C09134=1237.357,-18.440,-39.557,-179.564,5.238,148.773
C09135=1237.362,-18.689,-39.544,-179.566,5.238,148.774
C09136=1237.367,-18.939,-39.530,-179.568,5.238,148.775
C09137=1237.372,-19.189,-39.516,-179.571,5.237,148.776
C09138=1237.378,-19.438,-39.502,-179.573,5.237,148.776
C09139=1237.382,-19.687,-39.488,-179.576,5.237,148.777
C09140=1237.387,-19.938,-39.475,-179.578,5.236,148.778
C09141=1237.393,-20.187,-39.461,-179.581,5.237,148.778
C09142=1237.398,-20.436,-39.447,-179.583,5.236,148.779
C09143=1237.402,-20.686,-39.434,-179.585,5.236,148.780
C09144=1237.408,-20.935,-39.420,-179.588,5.236,148.780
C09145=1237.413,-21.185,-39.406,-179.591,5.235,148.781
C09146=1237.418,-21.435,-39.392,-179.593,5.236,148.782
C09147=1237.423,-21.684,-39.379,-179.596,5.236,148.783
C09148=1237.428,-21.954,-39.364,-179.598,5.235,148.783
C09149=1237.434,-22.223,-39.349,-179.601,5.235,148.784
C09150=1237.439,-22.492,-39.334,-179.604,5.235,148.785
C09151=1237.445,-22.761,-39.319,-179.606,5.235,148.786
C09152=1237.449,-23.010,-39.305,-179.609,5.234,148.786
C09153=1237.455,-23.261,-39.292,-179.611,5.234,148.787
C09154=1237.460,-23.510,-39.278,-179.614,5.234,148.788
C09155=1237.464,-23.759,-39.264,-179.616,5.234,148.789
C09156=1237.470,-24.009,-39.251,-179.619,5.234,148.789
C09157=1237.475,-24.259,-39.237,-179.621,5.233,148.790
C09158=1237.480,-24.509,-39.224,-179.623,5.234,148.791
C09159=1237.485,-24.758,-39.210,-179.626,5.233,148.791
C09160=1237.490,-25.007,-39.196,-179.628,5.234,148.792
C09161=1237.495,-25.257,-39.183,-179.631,5.233,148.793
C09162=1237.500,-25.506,-39.169,-179.634,5.233,148.794
C09163=1237.506,-25.757,-39.155,-179.636,5.233,148.794
C09164=1237.510,-26.005,-39.142,-179.639,5.232,148.795
C09165=1237.516,-26.256,-39.128,-179.641,5.233,148.796
C09166=1237.521,-26.504,-39.115,-179.643,5.232,148.796
C09167=1237.526,-26.755,-39.101,-179.646,5.232,148.797
C09168=1237.531,-27.004,-39.087,-179.648,5.232,148.798
C09169=1237.536,-27.253,-39.074,-179.651,5.232,148.799
C09170=1237.541,-27.503,-39.060,-179.653,5.232,148.799
C09171=1237.546,-27.752,-39.047,-179.655,5.231,148.800
C09172=1237.551,-28.002,-39.033,-179.658,5.231,148.801
C09173=1237.557,-28.252,-39.020,-179.661,5.231,148.802
C09174=1237.561,-28.502,-39.006,-179.663,5.231,148.802
C09175=1237.567,-28.751,-38.993,-179.665,5.231,148.803
C09176=1237.571,-29.001,-38.980,-179.668,5.231,148.804
C09177=1237.576,-29.251,-38.966,-179.671,5.230,148.804
C09178=1237.581,-29.500,-38.953,-179.673,5.231,148.805
C09179=1237.586,-29.750,-38.939,-179.675,5.230,148.806
C09180=1237.591,-29.999,-38.926,-179.678,5.230,148.806
C09181=1237.597,-30.249,-38.912,-179.680,5.230,148.807
C09182=1237.601,-30.498,-38.899,-179.683,5.229,148.808
C09183=1237.607,-30.748,-38.885,-179.685,5.230,148.809
C09184=1237.612,-30.998,-38.872,-179.688,5.229,148.809
C09185=1237.617,-31.247,-38.859,-179.690,5.230,148.810
C09186=1237.623,-31.497,-38.845,-179.693,5.229,148.811
C09187=1237.627,-31.746,-38.832,-179.696,5.229,148.812
C09188=1237.633,-31.996,-38.818,-179.698,5.229,148.812
C09189=1237.637,-32.246,-38.805,-179.700,5.229,148.813
C09190=1237.643,-32.495,-38.792,-179.702,5.229,148.814
C09191=1237.647,-32.745,-38.779,-179.705,5.228,148.814
C09192=1237.652,-32.994,-38.766,-179.708,5.228,148.815
C09193=1237.657,-33.244,-38.752,-179.710,5.228,148.816
C09194=1237.662,-33.493,-38.739,-179.712,5.228,148.816
C09195=1237.668,-33.743,-38.726,-179.715,5.228,148.817
C09196=1237.672,-33.992,-38.712,-179.717,5.227,148.818
C09197=1237.678,-34.242,-38.699,-179.720,5.227,148.819
C09198=1237.683,-34.492,-38.686,-179.722,5.228,148.819
C09199=1237.688,-34.741,-38.672,-179.725,5.227,148.820
C09200=1237.693,-34.991,-38.659,-179.727,5.227,148.821
C09201=1237.699,-35.240,-38.646,-179.730,5.227,148.822
C09202=1237.703,-35.490,-38.633,-179.732,5.227,148.822
C09203=1237.708,-35.739,-38.620,-179.735,5.227,148.823
C09204=1237.713,-35.989,-38.606,-179.737,5.226,148.824
C09205=1237.719,-36.239,-38.594,-179.739,5.227,148.824
C09206=1237.724,-36.489,-38.580,-179.742,5.226,148.825
C09207=1237.729,-36.738,-38.567,-179.744,5.226,148.826
C09208=1237.734,-36.987,-38.554,-179.747,5.226,148.826
C09209=1237.739,-37.237,-38.541,-179.749,5.226,148.827
C09210=1237.744,-37.487,-38.528,-179.752,5.226,148.828
C09211=1237.749,-37.737,-38.514,-179.755,5.225,148.829
C09212=1237.754,-37.986,-38.501,-179.757,5.226,148.829
C09213=1237.759,-38.236,-38.488,-179.759,5.225,148.830
C09214=1237.765,-38.485,-38.475,-179.761,5.226,148.831
C09215=1237.770,-38.735,-38.462,-179.764,5.225,148.832
C09216=1237.774,-38.985,-38.449,-179.766,5.225,148.832
C09217=1237.780,-39.234,-38.435,-179.769,5.225,148.833
C09218=1237.784,-39.484,-38.422,-179.772,5.224,148.834
C09219=1237.790,-39.733,-38.409,-179.774,5.225,148.834
C09220=1237.795,-39.983,-38.397,-179.776,5.224,148.835
C09221=1237.800,-40.233,-38.384,-179.778,5.225,148.836
C09222=1237.805,-40.482,-38.371,-179.782,5.224,148.837
C09223=1237.811,-40.732,-38.358,-179.784,5.225,148.837
C09224=1237.815,-40.982,-38.345,-179.786,5.224,148.838
C09225=1237.820,-41.230,-38.332,-179.789,5.224,148.839
C09226=1237.825,-41.481,-38.318,-179.791,5.224,148.840
C09227=1237.831,-41.730,-38.305,-179.794,5.224,148.840
C09228=1237.836,-41.979,-38.293,-179.796,5.224,148.841
C09229=1237.841,-42.230,-38.279,-179.798,5.223,148.842
C09230=1237.846,-42.479,-38.267,-179.801,5.224,148.842
C09231=1237.851,-42.728,-38.254,-179.803,5.223,148.843
C09232=1237.856,-42.978,-38.241,-179.806,5.223,148.844
C09233=1237.862,-43.228,-38.228,-179.808,5.223,148.844
C09234=1237.867,-43.477,-38.215,-179.811,5.223,148.845
C09235=1237.871,-43.727,-38.202,-179.813,5.223,148.846
C09236=1237.876,-43.977,-38.190,-179.816,5.223,148.847
C09237=1237.882,-44.226,-38.177,-179.818,5.223,148.847
C09238=1237.887,-44.476,-38.164,-179.821,5.222,148.848
C09239=1237.892,-44.726,-38.151,-179.823,5.222,148.849
C09240=1237.897,-44.975,-38.138,-179.825,5.222,148.850
C09241=1237.902,-45.225,-38.125,-179.828,5.222,148.850
C09242=1237.907,-45.475,-38.112,-179.830,5.222,148.851
C09243=1237.912,-45.724,-38.100,-179.833,5.222,148.852
C09244=1237.917,-45.974,-38.087,-179.835,5.222,148.852
C09245=1237.922,-46.223,-38.074,-179.838,5.221,148.853
C09246=1237.928,-46.473,-38.061,-179.840,5.222,148.854
C09247=1237.932,-46.723,-38.048,-179.843,5.222,148.855
C09248=1237.938,-46.972,-38.035,-179.845,5.221,148.855
C09249=1237.943,-47.221,-38.023,-179.848,5.221,148.856
C09250=1237.948,-47.471,-38.010,-179.850,5.221,148.857
C09251=1237.953,-47.721,-37.997,-179.852,5.221,148.858
C09252=1237.959,-47.990,-37.983,-179.855,5.221,148.858
C09253=1237.964,-48.260,-37.970,-179.858,5.221,148.859
C09254=1237.970,-48.531,-37.956,-179.860,5.221,148.860
C09255=1237.975,-48.800,-37.943,-179.863,5.220,148.861
C09256=1237.980,-49.050,-37.930,-179.865,5.221,148.861
C09257=1237.985,-49.299,-37.917,-179.868,5.220,148.862
C09258=1237.991,-49.549,-37.904,-179.870,5.220,148.863
C09259=1237.996,-49.798,-37.891,-179.873,5.220,148.864
C09260=1238.001,-50.048,-37.878,-179.876,5.220,148.864
C09261=1238.006,-50.297,-37.866,-179.878,5.220,148.865
C09262=1238.011,-50.547,-37.854,-179.880,5.220,148.866
C09263=1238.016,-50.796,-37.841,-179.882,5.220,148.866
C09264=1238.021,-51.046,-37.828,-179.885,5.220,148.867
C09265=1238.026,-51.296,-37.816,-179.887,5.220,148.868
C09266=1238.031,-51.545,-37.803,-179.890,5.219,148.869
C09267=1238.037,-51.795,-37.791,-179.892,5.220,148.869
C09268=1238.042,-52.045,-37.778,-179.895,5.219,148.870
C09269=1238.047,-52.295,-37.765,-179.897,5.219,148.871
C09270=1238.052,-52.544,-37.752,-179.899,5.219,148.871
C09271=1238.057,-52.793,-37.740,-179.902,5.219,148.872
C09272=1238.062,-53.044,-37.728,-179.905,5.219,148.873
C09273=1238.067,-53.293,-37.715,-179.907,5.219,148.874
C09274=1238.072,-53.543,-37.702,-179.909,5.219,148.874
C09275=1238.077,-53.792,-37.690,-179.912,5.219,148.875
C09276=1238.083,-54.042,-37.678,-179.914,5.219,148.876
C09277=1238.087,-54.292,-37.665,-179.917,5.218,148.877
C09278=1238.092,-54.541,-37.652,-179.919,5.219,148.877
C09279=1238.097,-54.790,-37.640,-179.922,5.218,148.878
C09280=1238.103,-55.040,-37.628,-179.924,5.219,148.879
C09281=1238.108,-55.290,-37.615,-179.926,5.218,148.879
C09282=1238.113,-55.540,-37.602,-179.928,5.218,148.880
C09283=1238.118,-55.790,-37.590,-179.931,5.218,148.881
C09284=1238.123,-56.039,-37.578,-179.934,5.217,148.881
C09285=1238.128,-56.288,-37.565,-179.936,5.218,148.882
C09286=1238.134,-56.538,-37.553,-179.939,5.218,148.883
C09287=1238.139,-56.788,-37.541,-179.941,5.218,148.884
C09288=1238.143,-57.038,-37.528,-179.944,5.218,148.885
C09289=1238.149,-57.288,-37.516,-179.946,5.218,148.885
C09290=1238.154,-57.537,-37.503,-179.948,5.217,148.886
C09291=1238.159,-57.786,-37.491,-179.951,5.218,148.887
C09292=1238.164,-58.036,-37.479,-179.953,5.217,148.887
C09293=1238.169,-58.285,-37.466,-179.955,5.218,148.888
C09294=1238.175,-58.535,-37.454,-179.958,5.217,148.889
C09295=1238.179,-58.785,-37.441,-179.960,5.217,148.889
C09296=1238.185,-59.035,-37.429,-179.963,5.217,148.890
C09297=1238.190,-59.285,-37.417,-179.965,5.217,148.891
C09298=1238.194,-59.534,-37.405,-179.968,5.217,148.892
C09299=1238.200,-59.784,-37.393,-179.971,5.217,148.892
C09300=1238.205,-60.033,-37.380,-179.973,5.217,148.893
C09301=1238.210,-60.283,-37.368,-179.975,5.216,148.894
C09302=1238.215,-60.532,-37.356,-179.977,5.217,148.895
C09303=1238.220,-60.782,-37.343,-179.980,5.216,148.895
C09304=1238.225,-61.032,-37.331,-179.982,5.217,148.896
C09305=1238.231,-61.281,-37.318,-179.985,5.216,148.897
C09306=1238.236,-61.531,-37.306,-179.987,5.216,148.897
C09307=1238.241,-61.781,-37.294,-179.990,5.216,148.898
C09308=1238.246,-62.030,-37.283,-179.992,5.216,148.899
C09309=1238.251,-62.280,-37.270,-179.994,5.216,148.900
C09310=1238.256,-62.530,-37.258,-179.997,5.216,148.900
C09311=1238.261,-62.779,-37.246,-179.999,5.216,148.901
C09312=1238.267,-63.029,-37.234,179.998,5.216,148.902
C09313=1238.272,-63.278,-37.221,179.996,5.216,148.903
C09314=1238.277,-63.529,-37.209,179.993,5.216,148.903
C09315=1238.282,-63.778,-37.197,179.991,5.216,148.904
C09316=1238.287,-64.028,-37.185,179.989,5.216,148.905
C09317=1238.292,-64.278,-37.173,179.986,5.216,148.905
C09318=1238.297,-64.527,-37.160,179.984,5.216,148.906
C09319=1238.303,-64.777,-37.149,179.981,5.215,148.907
C09320=1238.308,-65.026,-37.136,179.979,5.216,148.908
C09321=1238.312,-65.276,-37.125,179.977,5.215,148.908
C09322=1238.318,-65.526,-37.113,179.974,5.216,148.909
C09323=1238.323,-65.775,-37.100,179.972,5.215,148.910
C09324=1238.328,-66.025,-37.088,179.970,5.215,148.910
C09325=1238.334,-66.274,-37.076,179.967,5.215,148.911
C09326=1238.338,-66.524,-37.064,179.964,5.215,148.912
C09327=1238.344,-66.774,-37.052,179.962,5.215,148.913
C09328=1238.349,-67.023,-37.040,179.959,5.215,148.913
C09329=1238.354,-67.273,-37.028,179.957,5.215,148.914
C09330=1238.360,-67.523,-37.016,179.954,5.215,148.915
C09331=1238.364,-67.772,-37.004,179.952,5.215,148.916
C09332=1238.370,-68.022,-36.992,179.950,5.214,148.916
C09333=1238.375,-68.272,-36.980,179.947,5.215,148.917
C09334=1238.380,-68.521,-36.968,179.945,5.214,148.918
C09335=1238.385,-68.771,-36.956,179.943,5.215,148.918
C09336=1238.390,-69.021,-36.945,179.940,5.214,148.919
C09337=1238.395,-69.270,-36.932,179.938,5.214,148.920
C09338=1238.400,-69.520,-36.921,179.935,5.214,148.921
C09339=1238.405,-69.770,-36.909,179.933,5.214,148.921
C09340=1238.411,-70.019,-36.896,179.931,5.214,148.922
C09341=1238.416,-70.269,-36.884,179.928,5.214,148.923
C09342=1238.421,-70.519,-36.873,179.926,5.214,148.923
C09343=1238.426,-70.769,-36.861,179.923,5.214,148.924
C09344=1238.431,-71.018,-36.849,179.921,5.214,148.925
C09345=1238.436,-71.268,-36.837,179.918,5.214,148.926
C09346=1238.441,-71.517,-36.825,179.916,5.214,148.926
C09347=1238.447,-71.767,-36.813,179.914,5.214,148.927
C09348=1238.452,-72.017,-36.801,179.911,5.214,148.928
C09349=1238.457,-72.266,-36.790,179.909,5.214,148.929
C09350=1238.462,-72.516,-36.778,179.906,5.214,148.929
C09351=1238.467,-72.766,-36.766,179.904,5.214,148.930
C09352=1238.472,-73.016,-36.755,179.901,5.213,148.931
C09353=1238.477,-73.265,-36.742,179.899,5.214,148.931
C09354=1238.483,-73.514,-36.730,179.897,5.213,148.932
C09355=1238.488,-73.764,-36.719,179.895,5.214,148.933
C09356=1238.493,-74.034,-36.706,179.891,5.213,148.934
C09357=1238.499,-74.305,-36.693,179.889,5.214,148.934
C09358=1238.505,-74.575,-36.681,179.887,5.213,148.935
C09359=1238.510,-74.845,-36.668,179.884,5.213,148.936
C09360=1238.516,-75.095,-36.656,179.881,5.214,148.937
C09361=1238.520,-75.344,-36.644,179.879,5.213,148.937
C09362=1238.525,-75.594,-36.633,179.877,5.213,148.938
C09363=1238.531,-75.844,-36.621,179.874,5.213,148.939
C09364=1238.536,-76.093,-36.610,179.872,5.213,148.940
C09365=1238.542,-76.343,-36.598,179.869,5.213,148.940
C09366=1238.546,-76.593,-36.587,179.867,5.213,148.941
C09367=1238.552,-76.843,-36.575,179.864,5.213,148.942
C09368=1238.557,-77.093,-36.563,179.862,5.213,148.942
C09369=1238.562,-77.342,-36.551,179.860,5.213,148.943
C09370=1238.567,-77.592,-36.540,179.858,5.213,148.944
C09371=1238.572,-77.842,-36.528,179.855,5.212,148.945
C09372=1238.577,-78.092,-36.516,179.853,5.213,148.945
C09373=1238.582,-78.340,-36.505,179.850,5.212,148.946
C09374=1238.588,-78.590,-36.493,179.848,5.213,148.947
C09375=1238.592,-78.840,-36.482,179.845,5.212,148.947
C09376=1238.598,-79.089,-36.470,179.843,5.213,148.948
C09377=1238.603,-79.339,-36.458,179.841,5.212,148.949
C09378=1238.608,-79.589,-36.447,179.839,5.212,148.950
C09379=1238.613,-79.839,-36.435,179.835,5.212,148.950
C09380=1238.619,-80.088,-36.424,179.833,5.213,148.951
C09381=1238.624,-80.338,-36.412,179.831,5.212,148.952
C09382=1238.629,-80.587,-36.401,179.829,5.213,148.953
C09383=1238.634,-80.837,-36.389,179.826,5.213,148.953
C09384=1238.639,-81.087,-36.377,179.824,5.212,148.954
C09385=1238.644,-81.337,-36.366,179.822,5.213,148.955
C09386=1238.650,-81.586,-36.355,179.819,5.212,148.955
C09387=1238.655,-81.836,-36.343,179.817,5.213,148.956
C09388=1238.660,-82.086,-36.332,179.814,5.212,148.957
C09389=1238.665,-82.336,-36.321,179.812,5.212,148.958
C09390=1238.670,-82.586,-36.309,179.809,5.212,148.958
C09391=1238.675,-82.835,-36.298,179.807,5.212,148.959
C09392=1238.681,-83.084,-36.286,179.805,5.212,148.960
C09393=1238.686,-83.334,-36.275,179.803,5.212,148.960
C09394=1238.691,-83.584,-36.263,179.800,5.212,148.961
C09395=1238.696,-83.834,-36.252,179.798,5.212,148.962
C09396=1238.701,-84.084,-36.240,179.795,5.212,148.963
C09397=1238.706,-84.333,-36.229,179.793,5.212,148.963
C09398=1238.711,-84.583,-36.218,179.790,5.212,148.964
C09399=1238.717,-84.833,-36.206,179.788,5.212,148.965
C09400=1238.722,-85.082,-36.195,179.786,5.211,148.965
C09401=1238.727,-85.332,-36.183,179.784,5.212,148.966
C09402=1238.732,-85.581,-36.172,179.781,5.211,148.967
C09403=1238.737,-85.831,-36.161,179.778,5.212,148.968
C09404=1238.742,-86.081,-36.149,179.776,5.212,148.968
C09405=1238.747,-86.331,-36.139,179.774,5.212,148.969
C09406=1238.753,-86.580,-36.127,179.771,5.211,148.970
C09407=1238.758,-86.830,-36.116,179.769,5.212,148.971
C09408=1238.763,-87.079,-36.104,179.766,5.211,148.971
C09409=1238.768,-87.329,-36.093,179.764,5.212,148.972
C09410=1238.774,-87.579,-36.082,179.761,5.211,148.973
C09411=1238.779,-87.829,-36.071,179.759,5.212,148.973
C09412=1238.784,-88.079,-36.059,179.757,5.212,148.974
C09413=1238.789,-88.328,-36.048,179.754,5.211,148.975
C09414=1238.794,-88.577,-36.037,179.752,5.212,148.976
C09415=1238.800,-88.828,-36.026,179.750,5.211,148.976
C09416=1238.804,-89.077,-36.015,179.748,5.212,148.977
C09417=1238.809,-89.327,-36.003,179.745,5.211,148.978
C09418=1238.815,-89.576,-35.992,179.743,5.212,148.978
C09419=1238.820,-89.826,-35.981,179.740,5.211,148.979
C09420=1238.825,-90.076,-35.970,179.738,5.211,148.980
C09421=1238.831,-90.325,-35.958,179.735,5.211,148.981
C09422=1238.836,-90.575,-35.948,179.733,5.211,148.981
C09423=1238.841,-90.825,-35.936,179.731,5.211,148.982
C09424=1238.846,-91.075,-35.925,179.729,5.211,148.983
C09425=1238.852,-91.325,-35.914,179.726,5.211,148.983
C09426=1238.856,-91.574,-35.903,179.724,5.211,148.984
C09427=1238.861,-91.824,-35.892,179.721,5.211,148.985
C09428=1238.867,-92.073,-35.880,179.719,5.211,148.986
C09429=1238.872,-92.323,-35.870,179.716,5.211,148.986
C09430=1238.877,-92.573,-35.858,179.714,5.211,148.987
C09431=1238.883,-92.823,-35.848,179.712,5.211,148.988
C09432=1238.888,-93.072,-35.836,179.709,5.211,148.988
C09433=1238.892,-93.322,-35.825,179.707,5.211,148.989
C09434=1238.898,-93.572,-35.815,179.705,5.211,148.990
C09435=1238.903,-93.822,-35.803,179.703,5.211,148.991
C09436=1238.908,-94.071,-35.792,179.700,5.211,148.991
C09437=1238.914,-94.321,-35.781,179.698,5.211,148.992
C09438=1238.918,-94.570,-35.770,179.695,5.210,148.993
C09439=1238.923,-94.821,-35.760,179.693,5.211,148.993
C09440=1238.929,-95.070,-35.748,179.690,5.210,148.994
C09441=1238.934,-95.319,-35.737,179.688,5.211,148.995
C09442=1238.939,-95.570,-35.726,179.685,5.211,148.996
C09443=1238.944,-95.819,-35.715,179.683,5.211,148.996
C09444=1238.950,-96.069,-35.704,179.680,5.211,148.997
C09445=1238.955,-96.319,-35.693,179.678,5.211,148.998
C09446=1238.960,-96.568,-35.683,179.676,5.211,148.999
C09447=1238.965,-96.818,-35.671,179.673,5.211,148.999
C09448=1238.971,-97.067,-35.661,179.671,5.211,149.000
C09449=1238.975,-97.317,-35.650,179.669,5.211,149.001
C09450=1238.981,-97.568,-35.639,179.667,5.211,149.001
C09451=1238.986,-97.817,-35.628,179.664,5.211,149.002
C09452=1238.991,-98.067,-35.617,179.662,5.211,149.003
C09453=1238.997,-98.316,-35.606,179.659,5.210,149.004
C09454=1239.002,-98.566,-35.596,179.657,5.211,149.004
C09455=1239.006,-98.816,-35.584,179.654,5.210,149.005
C09456=1239.013,-99.065,-35.574,179.652,5.211,149.006
C09457=1239.017,-99.315,-35.562,179.650,5.210,149.006
C09458=1239.023,-99.565,-35.552,179.648,5.211,149.007
C09459=1239.028,-99.814,-35.541,179.645,5.211,149.008
C09460=1239.033,-100.085,-35.528,179.643,5.211,149.009
C09461=1239.039,-100.356,-35.518,179.640,5.210,149.009
C09462=1239.045,-100.627,-35.506,179.638,5.210,149.010
C09463=1239.050,-100.897,-35.494,179.635,5.210,149.011
C09464=1239.056,-101.147,-35.483,179.633,5.211,149.012
C09465=1239.061,-101.398,-35.473,179.630,5.210,149.012
C09466=1239.066,-101.647,-35.462,179.628,5.211,149.013
C09467=1239.071,-101.897,-35.451,179.625,5.210,149.014
C09468=1239.076,-102.146,-35.440,179.623,5.211,149.015
C09469=1239.082,-102.396,-35.430,179.621,5.210,149.015
C09470=1239.087,-102.646,-35.419,179.618,5.210,149.016
C09471=1239.092,-102.895,-35.408,179.616,5.211,149.017
C09472=1239.097,-103.145,-35.398,179.614,5.210,149.017
C09473=1239.102,-103.394,-35.387,179.612,5.211,149.018
C09474=1239.107,-103.645,-35.376,179.609,5.210,149.019
C09475=1239.113,-103.894,-35.366,179.607,5.211,149.020
C09476=1239.117,-104.144,-35.355,179.604,5.210,149.020
C09477=1239.122,-104.394,-35.344,179.602,5.211,149.021
C09478=1239.128,-104.643,-35.334,179.599,5.210,149.022
C09479=1239.133,-104.893,-35.322,179.597,5.210,149.022
C09480=1239.138,-105.143,-35.312,179.595,5.210,149.023
C09481=1239.143,-105.393,-35.302,179.592,5.210,149.024
C09482=1239.149,-105.642,-35.291,179.590,5.210,149.025
C09483=1239.154,-105.892,-35.280,179.588,5.210,149.025
C09484=1239.159,-106.142,-35.270,179.586,5.211,149.026
C09485=1239.164,-106.392,-35.259,179.583,5.210,149.027
C09486=1239.169,-106.641,-35.249,179.581,5.211,149.027
C09487=1239.174,-106.891,-35.238,179.578,5.210,149.028
C09488=1239.180,-107.141,-35.228,179.576,5.210,149.029
C09489=1239.185,-107.391,-35.217,179.574,5.210,149.029
C09490=1239.190,-107.640,-35.206,179.572,5.210,149.030
C09491=1239.195,-107.890,-35.196,179.569,5.210,149.031
C09492=1239.201,-108.139,-35.185,179.567,5.210,149.031
C09493=1239.206,-108.390,-35.175,179.565,5.210,149.032
C09494=1239.211,-108.639,-35.164,179.562,5.210,149.033
C09495=1239.217,-108.888,-35.154,179.560,5.210,149.034
C09496=1239.222,-109.138,-35.143,179.557,5.210,149.034
C09497=1239.227,-109.388,-35.133,179.555,5.210,149.035
C09498=1239.232,-109.638,-35.122,179.553,5.210,149.036
C09499=1239.238,-109.887,-35.111,179.551,5.210,149.036
C09500=1239.243,-110.137,-35.101,179.548,5.210,149.037
C09501=1239.248,-110.387,-35.091,179.546,5.210,149.038
C09502=1239.253,-110.637,-35.081,179.543,5.209,149.039
C09503=1239.258,-110.886,-35.070,179.541,5.210,149.039
C09504=1239.263,-111.137,-35.060,179.539,5.210,149.040
C09505=1239.269,-111.386,-35.050,179.536,5.210,149.041
C09506=1239.274,-111.635,-35.039,179.534,5.210,149.041
C09507=1239.279,-111.885,-35.028,179.532,5.210,149.042
C09508=1239.285,-112.135,-35.018,179.529,5.210,149.043
C09509=1239.290,-112.385,-35.007,179.527,5.210,149.044
C09510=1239.295,-112.635,-34.997,179.525,5.210,149.044
C09511=1239.300,-112.884,-34.988,179.522,5.209,149.045
C09512=1239.305,-113.134,-34.977,179.520,5.210,149.046
C09513=1239.311,-113.384,-34.967,179.518,5.210,149.046
C09514=1239.316,-113.634,-34.956,179.515,5.210,149.047
C09515=1239.321,-113.884,-34.946,179.513,5.210,149.048
C09516=1239.327,-114.132,-34.935,179.510,5.210,149.049
C09517=1239.332,-114.383,-34.925,179.508,5.210,149.049
C09518=1239.336,-114.632,-34.915,179.506,5.210,149.050
C09519=1239.341,-114.882,-34.904,179.503,5.210,149.051
C09520=1239.347,-115.132,-34.894,179.501,5.210,149.051
C09521=1239.353,-115.381,-34.884,179.499,5.210,149.052
C09522=1239.358,-115.632,-34.873,179.497,5.210,149.053
C09523=1239.363,-115.881,-34.863,179.494,5.209,149.053
C09524=1239.368,-116.131,-34.853,179.492,5.210,149.054
C09525=1239.373,-116.381,-34.843,179.490,5.209,149.055
C09526=1239.379,-116.630,-34.833,179.488,5.210,149.056
C09527=1239.384,-116.880,-34.822,179.485,5.209,149.056
C09528=1239.389,-117.130,-34.813,179.483,5.210,149.057
C09529=1239.394,-117.379,-34.802,179.480,5.209,149.058
C09530=1239.399,-117.629,-34.792,179.478,5.210,149.058
C09531=1239.405,-117.879,-34.782,179.476,5.210,149.059
C09532=1239.410,-118.128,-34.771,179.473,5.210,149.060
C09533=1239.415,-118.378,-34.761,179.471,5.210,149.061
C09534=1239.420,-118.628,-34.751,179.468,5.209,149.061
C09535=1239.426,-118.877,-34.741,179.466,5.210,149.062
C09536=1239.431,-119.128,-34.730,179.464,5.209,149.063
C09537=1239.436,-119.378,-34.721,179.462,5.210,149.063
C09538=1239.442,-119.627,-34.711,179.459,5.209,149.064
C09539=1239.447,-119.877,-34.701,179.457,5.210,149.065
C09540=1239.451,-120.127,-34.691,179.455,5.210,149.066
C09541=1239.457,-120.376,-34.681,179.452,5.210,149.066
C09542=1239.462,-120.626,-34.670,179.450,5.210,149.067
C09543=1239.468,-120.876,-34.660,179.448,5.209,149.067
C09544=1239.473,-121.125,-34.650,179.446,5.210,149.068
C09545=1239.478,-121.375,-34.640,179.443,5.209,149.069
C09546=1239.483,-121.626,-34.630,179.441,5.209,149.070
C09547=1239.488,-121.875,-34.621,179.438,5.209,149.070
C09548=1239.493,-122.125,-34.610,179.436,5.209,149.071
C09549=1239.499,-122.375,-34.600,179.434,5.210,149.072
C09550=1239.504,-122.624,-34.590,179.431,5.209,149.072
C09551=1239.509,-122.873,-34.580,179.429,5.210,149.073
C09552=1239.514,-123.124,-34.570,179.427,5.209,149.074
C09553=1239.519,-123.373,-34.561,179.424,5.210,149.075
C09554=1239.525,-123.623,-34.551,179.422,5.209,149.075
C09555=1239.530,-123.873,-34.540,179.420,5.210,149.076
C09556=1239.535,-124.122,-34.530,179.417,5.209,149.077
C09557=1239.541,-124.372,-34.520,179.415,5.209,149.077
C09558=1239.546,-124.622,-34.511,179.413,5.210,149.078
C09559=1239.551,-124.872,-34.501,179.411,5.209,149.079
C09560=1239.556,-125.122,-34.490,179.408,5.209,149.079
C09561=1239.562,-125.371,-34.480,179.406,5.209,149.080
C09562=1239.567,-125.621,-34.471,179.404,5.209,149.081
C09563=1239.572,-125.871,-34.461,179.401,5.209,149.082
C09564=1239.151,-125.882,-34.496,179.397,5.212,149.084
C09565=1239.145,-125.632,-34.505,179.399,5.213,149.083
C09566=1239.139,-125.382,-34.515,179.401,5.213,149.082
C09567=1239.135,-125.132,-34.525,179.404,5.213,149.082
C09568=1239.129,-124.883,-34.536,179.406,5.213,149.081
C09569=1239.124,-124.633,-34.545,179.409,5.213,149.080
C09570=1239.119,-124.383,-34.555,179.411,5.213,149.079
C09571=1239.114,-124.133,-34.565,179.413,5.212,149.079
C09572=1239.109,-123.884,-34.575,179.416,5.213,149.078
C09573=1239.103,-123.634,-34.585,179.418,5.212,149.077
C09574=1239.098,-123.383,-34.595,179.420,5.213,149.077
C09575=1239.093,-123.134,-34.605,179.422,5.213,149.076
C09576=1239.087,-122.884,-34.615,179.425,5.213,149.075
C09577=1239.082,-122.635,-34.625,179.427,5.213,149.075
C09578=1239.078,-122.385,-34.635,179.429,5.212,149.074
C09579=1239.072,-122.135,-34.645,179.432,5.213,149.073
C09580=1239.066,-121.885,-34.655,179.434,5.213,149.072
C09581=1239.062,-121.635,-34.665,179.436,5.213,149.072
C09582=1239.056,-121.386,-34.675,179.438,5.213,149.071
C09583=1239.051,-121.136,-34.685,179.441,5.213,149.070
C09584=1239.046,-120.887,-34.695,179.443,5.213,149.070
C09585=1239.041,-120.637,-34.705,179.446,5.213,149.069
C09586=1239.035,-120.387,-34.716,179.448,5.213,149.068
C09587=1239.030,-120.138,-34.726,179.450,5.212,149.067
C09588=1239.025,-119.887,-34.735,179.453,5.213,149.067
C09589=1239.019,-119.638,-34.745,179.454,5.213,149.066
C09590=1239.014,-119.388,-34.755,179.457,5.213,149.066
C09591=1239.010,-119.138,-34.765,179.459,5.213,149.065
C09592=1239.004,-118.889,-34.776,179.462,5.213,149.064
C09593=1238.998,-118.639,-34.786,179.464,5.213,149.063
C09594=1238.993,-118.389,-34.796,179.467,5.213,149.063
C09595=1238.988,-118.140,-34.806,179.469,5.213,149.062
C09596=1238.983,-117.890,-34.816,179.471,5.213,149.061
C09597=1238.978,-117.640,-34.827,179.473,5.213,149.061
C09598=1238.972,-117.390,-34.837,179.476,5.213,149.060
C09599=1238.967,-117.141,-34.847,179.478,5.213,149.059
C09600=1238.962,-116.891,-34.857,179.480,5.213,149.058
C09601=1238.957,-116.641,-34.867,179.483,5.213,149.058
C09602=1238.952,-116.391,-34.878,179.485,5.213,149.057
C09603=1238.946,-116.141,-34.888,179.488,5.213,149.056
C09604=1238.941,-115.892,-34.898,179.490,5.213,149.055
C09605=1238.936,-115.642,-34.908,179.492,5.213,149.055
C09606=1238.931,-115.392,-34.919,179.495,5.213,149.054
C09607=1238.925,-115.143,-34.929,179.497,5.213,149.053
C09608=1238.920,-114.893,-34.939,179.499,5.213,149.053
C09609=1238.915,-114.643,-34.949,179.501,5.213,149.052
C09610=1238.910,-114.393,-34.960,179.504,5.214,149.051
C09611=1238.905,-114.144,-34.970,179.506,5.213,149.051
C09612=1238.899,-113.894,-34.980,179.509,5.214,149.050
C09613=1238.894,-113.644,-34.991,179.511,5.213,149.049
C09614=1238.888,-113.394,-35.001,179.513,5.213,149.049
C09615=1238.883,-113.145,-35.011,179.515,5.213,149.048
C09616=1238.879,-112.895,-35.021,179.517,5.213,149.047
C09617=1238.873,-112.645,-35.031,179.520,5.213,149.046
C09618=1238.868,-112.396,-35.042,179.522,5.213,149.046
C09619=1238.863,-112.146,-35.053,179.525,5.213,149.045
C09620=1238.858,-111.896,-35.063,179.527,5.213,149.044
C09621=1238.852,-111.646,-35.073,179.530,5.214,149.044
C09622=1238.847,-111.397,-35.084,179.532,5.213,149.043
C09623=1238.842,-111.146,-35.094,179.534,5.213,149.042
C09624=1238.837,-110.897,-35.104,179.537,5.213,149.041
C09625=1238.832,-110.647,-35.114,179.539,5.213,149.041
C09626=1238.826,-110.398,-35.125,179.541,5.213,149.040
C09627=1238.821,-110.148,-35.136,179.543,5.213,149.039
C09628=1238.816,-109.898,-35.146,179.546,5.213,149.039
C09629=1238.810,-109.649,-35.156,179.548,5.213,149.038
C09630=1238.805,-109.399,-35.167,179.551,5.214,149.037
C09631=1238.800,-109.149,-35.177,179.553,5.213,149.036
C09632=1238.795,-108.899,-35.188,179.556,5.214,149.036
C09633=1238.789,-108.650,-35.199,179.558,5.213,149.035
C09634=1238.784,-108.400,-35.209,179.560,5.213,149.034
C09635=1238.779,-108.150,-35.219,179.563,5.213,149.034
C09636=1238.774,-107.900,-35.231,179.565,5.213,149.033
C09637=1238.768,-107.651,-35.241,179.567,5.213,149.032
C09638=1238.763,-107.401,-35.251,179.569,5.213,149.031
C09639=1238.758,-107.151,-35.262,179.572,5.214,149.031
C09640=1238.754,-106.901,-35.272,179.574,5.213,149.030
C09641=1238.748,-106.652,-35.283,179.576,5.214,149.029
C09642=1238.743,-106.402,-35.293,179.578,5.214,149.029
C09643=1238.738,-106.152,-35.303,179.581,5.214,149.028
C09644=1238.733,-105.903,-35.315,179.583,5.214,149.027
C09645=1238.727,-105.653,-35.325,179.585,5.213,149.027
C09646=1238.722,-105.403,-35.335,179.588,5.214,149.026
C09647=1238.717,-105.153,-35.346,179.590,5.213,149.025
C09648=1238.712,-104.904,-35.357,179.593,5.214,149.024
C09649=1238.707,-104.654,-35.367,179.595,5.214,149.024
C09650=1238.702,-104.404,-35.378,179.598,5.214,149.023
C09651=1238.696,-104.155,-35.389,179.600,5.214,149.022
C09652=1238.690,-103.905,-35.400,179.602,5.214,149.022
C09653=1238.685,-103.655,-35.410,179.604,5.214,149.021
C09654=1238.680,-103.405,-35.421,179.607,5.214,149.020
C09655=1238.675,-103.156,-35.432,179.609,5.214,149.019
C09656=1238.670,-102.906,-35.442,179.611,5.213,149.019
C09657=1238.664,-102.657,-35.453,179.614,5.214,149.018
C09658=1238.659,-102.406,-35.464,179.616,5.214,149.017
C09659=1238.655,-102.157,-35.475,179.619,5.214,149.017
C09660=1238.649,-101.907,-35.485,179.621,5.214,149.016
C09661=1238.644,-101.657,-35.496,179.623,5.214,149.015
C09662=1238.639,-101.408,-35.507,179.626,5.214,149.014
C09663=1238.634,-101.158,-35.517,179.628,5.214,149.014
C09664=1238.628,-100.909,-35.528,179.630,5.214,149.013
C09665=1238.623,-100.637,-35.540,179.634,5.214,149.012
C09666=1238.618,-100.367,-35.551,179.636,5.214,149.011
C09667=1238.611,-100.096,-35.563,179.638,5.214,149.011
C09668=1238.606,-99.825,-35.575,179.640,5.214,149.010
C09669=1238.601,-99.575,-35.586,179.643,5.214,149.009
C09670=1238.595,-99.326,-35.596,179.645,5.214,149.009
C09671=1238.591,-99.076,-35.607,179.648,5.214,149.008
C09672=1238.586,-98.826,-35.618,179.650,5.214,149.007
C09673=1238.580,-98.577,-35.629,179.653,5.214,149.006
C09674=1238.575,-98.327,-35.640,179.655,5.214,149.006
C09675=1238.569,-98.077,-35.651,179.657,5.214,149.005
C09676=1238.564,-97.827,-35.662,179.659,5.214,149.004
C09677=1238.560,-97.577,-35.673,179.662,5.214,149.004
C09678=1238.554,-97.328,-35.683,179.664,5.214,149.003
C09679=1238.549,-97.078,-35.694,179.667,5.215,149.002
C09680=1238.544,-96.829,-35.705,179.669,5.214,149.001
C09681=1238.538,-96.579,-35.717,179.671,5.214,149.001
C09682=1238.533,-96.329,-35.727,179.674,5.214,149.000
C09683=1238.528,-96.080,-35.738,179.676,5.214,148.999
C09684=1238.523,-95.829,-35.749,179.679,5.214,148.999
C09685=1238.518,-95.580,-35.760,179.681,5.214,148.998
C09686=1238.512,-95.330,-35.771,179.683,5.215,148.997
C09687=1238.507,-95.080,-35.782,179.685,5.214,148.996
C09688=1238.502,-94.831,-35.793,179.688,5.215,148.996
C09689=1238.497,-94.581,-35.804,179.690,5.214,148.995
C09690=1238.492,-94.332,-35.815,179.693,5.215,148.994
C09691=1238.486,-94.082,-35.826,179.695,5.214,148.994
C09692=1238.481,-93.832,-35.837,179.698,5.215,148.993
C09693=1238.476,-93.582,-35.848,179.700,5.215,148.992
C09694=1238.471,-93.333,-35.858,179.702,5.215,148.991
C09695=1238.465,-93.083,-35.870,179.705,5.214,148.990
C09696=1238.460,-92.833,-35.881,179.708,5.215,148.990
C09697=1238.455,-92.584,-35.892,179.710,5.214,148.989
C09698=1238.450,-92.334,-35.903,179.712,5.214,148.988
C09699=1238.445,-92.084,-35.914,179.715,5.214,148.988
C09700=1238.439,-91.835,-35.925,179.717,5.214,148.987
C09701=1238.435,-91.585,-35.936,179.719,5.215,148.986
C09702=1238.429,-91.334,-35.948,179.721,5.214,148.986
C09703=1238.424,-91.086,-35.959,179.724,5.215,148.985
C09704=1238.419,-90.836,-35.970,179.726,5.214,148.984
C09705=1238.414,-90.586,-35.980,179.729,5.215,148.983
C09706=1238.409,-90.336,-35.992,179.731,5.214,148.983
C09707=1238.403,-90.087,-36.003,179.734,5.215,148.982
C09708=1238.399,-89.837,-36.015,179.736,5.215,148.981
C09709=1238.393,-89.587,-36.026,179.738,5.215,148.981
C09710=1238.388,-89.338,-36.037,179.740,5.215,148.980
C09711=1238.383,-89.088,-36.048,179.743,5.215,148.979
C09712=1238.377,-88.838,-36.060,179.745,5.215,148.978
C09713=1238.372,-88.588,-36.070,179.748,5.215,148.978
C09714=1238.367,-88.339,-36.081,179.750,5.215,148.977
C09715=1238.362,-88.089,-36.093,179.753,5.215,148.976
C09716=1238.357,-87.839,-36.104,179.755,5.215,148.976
C09717=1238.352,-87.589,-36.115,179.757,5.215,148.975
C09718=1238.346,-87.340,-36.127,179.760,5.215,148.974
C09719=1238.341,-87.090,-36.138,179.762,5.215,148.973
C09720=1238.337,-86.841,-36.149,179.764,5.215,148.973
C09721=1238.331,-86.591,-36.161,179.766,5.215,148.972
C09722=1238.326,-86.341,-36.171,179.769,5.215,148.971
C09723=1238.320,-86.091,-36.183,179.771,5.215,148.971
C09724=1238.316,-85.842,-36.194,179.774,5.215,148.970
C09725=1238.311,-85.592,-36.206,179.776,5.215,148.969
C09726=1238.305,-85.343,-36.217,179.779,5.216,148.968
C09727=1238.300,-85.093,-36.228,179.781,5.215,148.968
C09728=1238.294,-84.843,-36.240,179.783,5.216,148.967
C09729=1238.290,-84.593,-36.251,179.785,5.215,148.966
C09730=1238.285,-84.343,-36.262,179.788,5.216,148.966
C09731=1238.279,-84.094,-36.274,179.791,5.215,148.965
C09732=1238.274,-83.844,-36.285,179.793,5.216,148.964
C09733=1238.269,-83.595,-36.297,179.795,5.215,148.963
C09734=1238.264,-83.345,-36.308,179.798,5.216,148.963
C09735=1238.259,-83.095,-36.320,179.800,5.215,148.962
C09736=1238.253,-82.845,-36.330,179.803,5.216,148.961
C09737=1238.248,-82.596,-36.342,179.805,5.215,148.960
C09738=1238.243,-82.346,-36.353,179.808,5.216,148.960
C09739=1238.238,-82.096,-36.365,179.810,5.216,148.959
C09740=1238.233,-81.846,-36.377,179.812,5.216,148.958
C09741=1238.228,-81.597,-36.388,179.815,5.216,148.958
C09742=1238.222,-81.347,-36.399,179.817,5.216,148.957
C09743=1238.217,-81.098,-36.411,179.819,5.216,148.956
C09744=1238.212,-80.848,-36.423,179.822,5.216,148.955
C09745=1238.207,-80.598,-36.434,179.824,5.216,148.955
C09746=1238.202,-80.348,-36.446,179.827,5.216,148.954
C09747=1238.197,-80.099,-36.457,179.829,5.216,148.953
C09748=1238.191,-79.849,-36.469,179.831,5.216,148.953
C09749=1238.186,-79.600,-36.480,179.834,5.216,148.952
C09750=1238.181,-79.350,-36.492,179.836,5.216,148.951
C09751=1238.176,-79.100,-36.503,179.838,5.216,148.950
C09752=1238.171,-78.850,-36.515,179.840,5.216,148.950
C09753=1238.166,-78.601,-36.526,179.843,5.216,148.949
C09754=1238.160,-78.351,-36.538,179.845,5.216,148.948
C09755=1238.156,-78.102,-36.549,179.848,5.216,148.947
C09756=1238.150,-77.852,-36.561,179.850,5.216,148.947
C09757=1238.145,-77.602,-36.572,179.853,5.216,148.946
C09758=1238.140,-77.352,-36.584,179.855,5.216,148.945
C09759=1238.135,-77.102,-36.596,179.858,5.216,148.945
C09760=1238.130,-76.853,-36.607,179.860,5.216,148.944
C09761=1238.124,-76.603,-36.619,179.863,5.217,148.943
C09762=1238.119,-76.354,-36.630,179.865,5.216,148.942
C09763=1238.114,-76.105,-36.643,179.867,5.217,148.942
C09764=1238.109,-75.855,-36.654,179.869,5.216,148.941
C09765=1238.104,-75.605,-36.666,179.872,5.217,148.940
C09766=1238.098,-75.355,-36.678,179.874,5.217,148.940
C09767=1238.094,-75.105,-36.689,179.877,5.217,148.939
C09768=1238.088,-74.856,-36.701,179.879,5.217,148.938
C09769=1238.082,-74.586,-36.714,179.882,5.217,148.937
C09770=1238.077,-74.316,-36.727,179.885,5.217,148.937
C09771=1238.072,-74.045,-36.740,179.887,5.217,148.936
C09772=1238.066,-73.775,-36.751,179.890,5.217,148.935
C09773=1238.060,-73.526,-36.764,179.892,5.217,148.934
C09774=1238.056,-73.276,-36.775,179.894,5.218,148.934
C09775=1238.050,-73.026,-36.787,179.897,5.217,148.933
C09776=1238.045,-72.776,-36.799,179.900,5.217,148.932
C09777=1238.040,-72.526,-36.810,179.902,5.217,148.931
C09778=1238.035,-72.277,-36.823,179.904,5.217,148.931
C09779=1238.030,-72.027,-36.835,179.906,5.217,148.930
C09780=1238.025,-71.778,-36.846,179.909,5.218,148.929
C09781=1238.020,-71.528,-36.858,179.911,5.217,148.929
C09782=1238.014,-71.278,-36.870,179.914,5.218,148.928
C09783=1238.010,-71.029,-36.882,179.916,5.217,148.927
C09784=1238.004,-70.779,-36.894,179.919,5.218,148.926
C09785=1237.999,-70.529,-36.906,179.921,5.218,148.926
C09786=1237.994,-70.279,-36.917,179.923,5.218,148.925
C09787=1237.989,-70.030,-36.930,179.926,5.218,148.924
C09788=1237.984,-69.780,-36.941,179.928,5.218,148.924
C09789=1237.978,-69.530,-36.953,179.930,5.218,148.923
C09790=1237.974,-69.280,-36.965,179.933,5.218,148.922
C09791=1237.968,-69.031,-36.977,179.935,5.218,148.921
C09792=1237.963,-68.781,-36.989,179.938,5.218,148.920
C09793=1237.958,-68.532,-37.000,179.940,5.218,148.920
C09794=1237.953,-68.282,-37.013,179.943,5.218,148.919
C09795=1237.948,-68.032,-37.025,179.945,5.218,148.918
C09796=1237.942,-67.782,-37.037,179.948,5.218,148.918
C09797=1237.938,-67.533,-37.049,179.950,5.219,148.917
C09798=1237.932,-67.283,-37.061,179.953,5.218,148.916
C09799=1237.927,-67.033,-37.073,179.955,5.219,148.916
C09800=1237.922,-66.784,-37.085,179.957,5.219,148.915
C09801=1237.916,-66.534,-37.097,179.960,5.219,148.914
C09802=1237.912,-66.285,-37.108,179.962,5.219,148.913
C09803=1237.907,-66.035,-37.121,179.965,5.219,148.913
C09804=1237.901,-65.785,-37.133,179.967,5.219,148.912
C09805=1237.896,-65.536,-37.145,179.969,5.219,148.911
C09806=1237.891,-65.286,-37.157,179.972,5.219,148.911
C09807=1237.886,-65.036,-37.169,179.974,5.220,148.910
C09808=1237.881,-64.787,-37.181,179.977,5.219,148.909
C09809=1237.875,-64.537,-37.193,179.979,5.219,148.908
C09810=1237.870,-64.288,-37.206,179.982,5.219,148.908
C09811=1237.865,-64.038,-37.218,179.984,5.219,148.907
C09812=1237.860,-63.789,-37.230,179.986,5.219,148.906
C09813=1237.855,-63.539,-37.241,179.989,5.220,148.905
C09814=1237.850,-63.289,-37.253,179.991,5.219,148.905
C09815=1237.845,-63.040,-37.266,179.994,5.220,148.904
C09816=1237.839,-62.790,-37.278,179.996,5.219,148.903
C09817=1237.834,-62.540,-37.290,179.998,5.220,148.903
C09818=1237.829,-62.290,-37.303,-179.999,5.220,148.902
C09819=1237.825,-62.041,-37.315,-179.997,5.220,148.901
C09820=1237.819,-61.791,-37.327,-179.995,5.220,148.900
C09821=1237.814,-61.542,-37.339,-179.992,5.220,148.900
C09822=1237.809,-61.292,-37.351,-179.990,5.220,148.899
C09823=1237.804,-61.042,-37.364,-179.987,5.220,148.898
C09824=1237.798,-60.792,-37.376,-179.985,5.220,148.897
C09825=1237.793,-60.543,-37.388,-179.982,5.220,148.897
C09826=1237.788,-60.294,-37.401,-179.979,5.221,148.896
C09827=1237.783,-60.044,-37.413,-179.977,5.220,148.895
C09828=1237.779,-59.794,-37.425,-179.975,5.221,148.895
C09829=1237.773,-59.544,-37.437,-179.972,5.221,148.894
C09830=1237.768,-59.295,-37.449,-179.970,5.221,148.893
C09831=1237.763,-59.045,-37.461,-179.968,5.221,148.892
C09832=1237.758,-58.796,-37.474,-179.965,5.221,148.892
C09833=1237.753,-58.546,-37.487,-179.963,5.221,148.891
C09834=1237.747,-58.296,-37.498,-179.960,5.221,148.890
C09835=1237.742,-58.047,-37.511,-179.958,5.221,148.890
C09836=1237.737,-57.796,-37.523,-179.956,5.221,148.889
C09837=1237.732,-57.547,-37.536,-179.953,5.221,148.888
C09838=1237.727,-57.298,-37.548,-179.950,5.221,148.887
C09839=1237.721,-57.048,-37.560,-179.948,5.221,148.887
C09840=1237.716,-56.799,-37.573,-179.946,5.221,148.886
C09841=1237.711,-56.549,-37.586,-179.943,5.221,148.885
C09842=1237.706,-56.299,-37.598,-179.941,5.222,148.885
C09843=1237.701,-56.049,-37.610,-179.938,5.222,148.884
C09844=1237.696,-55.800,-37.623,-179.936,5.222,148.883
C09845=1237.691,-55.550,-37.635,-179.933,5.222,148.882
C09846=1237.686,-55.301,-37.648,-179.931,5.222,148.882
C09847=1237.680,-55.051,-37.660,-179.929,5.222,148.881
C09848=1237.676,-54.801,-37.672,-179.927,5.222,148.880
C09849=1237.671,-54.551,-37.685,-179.924,5.223,148.880
C09850=1237.665,-54.302,-37.698,-179.921,5.222,148.879
C09851=1237.660,-54.052,-37.709,-179.919,5.222,148.878
C09852=1237.655,-53.803,-37.722,-179.916,5.222,148.877
C09853=1237.650,-53.553,-37.735,-179.914,5.223,148.877
C09854=1237.645,-53.303,-37.748,-179.912,5.222,148.876
C09855=1237.640,-53.054,-37.760,-179.909,5.223,148.875
C09856=1237.635,-52.804,-37.772,-179.906,5.223,148.874
C09857=1237.630,-52.555,-37.785,-179.904,5.223,148.874
C09858=1237.625,-52.305,-37.798,-179.902,5.223,148.873
C09859=1237.620,-52.055,-37.810,-179.900,5.223,148.872
C09860=1237.614,-51.806,-37.822,-179.897,5.224,148.872
C09861=1237.609,-51.556,-37.835,-179.895,5.223,148.871
C09862=1237.605,-51.306,-37.848,-179.892,5.224,148.870
C09863=1237.600,-51.057,-37.860,-179.890,5.223,148.869
C09864=1237.593,-50.807,-37.873,-179.887,5.224,148.869
C09865=1237.588,-50.557,-37.885,-179.885,5.223,148.868
C09866=1237.584,-50.307,-37.898,-179.882,5.224,148.867
C09867=1237.579,-50.058,-37.911,-179.879,5.224,148.866
C09868=1237.574,-49.809,-37.924,-179.877,5.224,148.866
C09869=1237.568,-49.559,-37.936,-179.875,5.224,148.865
C09870=1237.564,-49.309,-37.949,-179.873,5.224,148.864
C09871=1237.559,-49.059,-37.961,-179.870,5.225,148.864
C09872=1237.553,-48.810,-37.974,-179.868,5.224,148.863
C09873=1237.548,-48.540,-37.988,-179.865,5.224,148.862
C09874=1237.542,-48.271,-38.001,-179.862,5.225,148.861
C09875=1237.536,-48.001,-38.015,-179.860,5.225,148.861
C09876=1237.531,-47.731,-38.029,-179.857,5.225,148.860
C09877=1237.526,-47.482,-38.042,-179.854,5.225,148.859
C09878=1237.521,-47.233,-38.054,-179.852,5.225,148.858
C09879=1237.516,-46.982,-38.068,-179.849,5.225,148.858
C09880=1237.511,-46.733,-38.081,-179.847,5.225,148.857
C09881=1237.505,-46.483,-38.092,-179.845,5.225,148.856
C09882=1237.500,-46.234,-38.105,-179.843,5.225,148.855
C09883=1237.496,-45.984,-38.118,-179.840,5.226,148.855
C09884=1237.490,-45.734,-38.131,-179.838,5.225,148.854
C09885=1237.485,-45.485,-38.144,-179.835,5.226,148.853
C09886=1237.480,-45.235,-38.157,-179.832,5.226,148.853
C09887=1237.475,-44.985,-38.169,-179.830,5.226,148.852
C09888=1237.470,-44.736,-38.182,-179.828,5.227,148.851
C09889=1237.465,-44.486,-38.196,-179.826,5.226,148.851
C09890=1237.459,-44.237,-38.208,-179.822,5.226,148.850
C09891=1237.454,-43.987,-38.221,-179.820,5.226,148.849
C09892=1237.450,-43.737,-38.234,-179.818,5.227,148.848
C09893=1237.444,-43.488,-38.247,-179.816,5.226,148.847
C09894=1237.439,-43.238,-38.259,-179.813,5.227,148.847
C09895=1237.434,-42.988,-38.272,-179.810,5.227,148.846
C09896=1237.429,-42.739,-38.285,-179.808,5.227,148.845
C09897=1237.423,-42.489,-38.298,-179.806,5.227,148.845
C09898=1237.419,-42.240,-38.312,-179.803,5.227,148.844
C09899=1237.414,-41.991,-38.325,-179.801,5.228,148.843
C09900=1237.408,-41.741,-38.338,-179.799,5.227,148.843
C09901=1237.404,-41.491,-38.351,-179.796,5.228,148.842
C09902=1237.398,-41.242,-38.363,-179.793,5.228,148.841
C09903=1237.394,-40.992,-38.376,-179.791,5.228,148.840
C09904=1237.388,-40.742,-38.389,-179.788,5.228,148.840
C09905=1237.383,-40.493,-38.402,-179.786,5.228,148.839
C09906=1237.378,-40.243,-38.415,-179.783,5.228,148.838
C09907=1237.373,-39.993,-38.428,-179.781,5.228,148.837
C09908=1237.368,-39.744,-38.442,-179.779,5.228,148.837
C09909=1237.363,-39.494,-38.455,-179.776,5.229,148.836
C09910=1237.357,-39.245,-38.468,-179.774,5.229,148.835
C09911=1237.353,-38.995,-38.481,-179.771,5.229,148.835
C09912=1237.348,-38.745,-38.493,-179.769,5.229,148.834
C09913=1237.342,-38.496,-38.506,-179.766,5.229,148.833
C09914=1237.337,-38.246,-38.519,-179.764,5.229,148.833
C09915=1237.333,-37.997,-38.533,-179.761,5.229,148.832
C09916=1237.327,-37.747,-38.546,-179.759,5.230,148.831
C09917=1237.322,-37.497,-38.559,-179.756,5.229,148.830
C09918=1237.316,-37.248,-38.572,-179.754,5.230,148.830
C09919=1237.312,-36.998,-38.585,-179.752,5.230,148.829
C09920=1237.307,-36.749,-38.598,-179.749,5.230,148.828
C09921=1237.302,-36.499,-38.612,-179.747,5.230,148.827
C09922=1237.297,-36.249,-38.625,-179.744,5.230,148.827
C09923=1237.291,-35.999,-38.638,-179.742,5.231,148.826
C09924=1237.286,-35.750,-38.651,-179.740,5.230,148.825
C09925=1237.281,-35.501,-38.664,-179.737,5.231,148.825
C09926=1237.276,-35.251,-38.678,-179.735,5.231,148.824
C09927=1237.271,-35.001,-38.690,-179.732,5.231,148.823
C09928=1237.266,-34.752,-38.704,-179.729,5.231,148.822
C09929=1237.261,-34.502,-38.717,-179.727,5.231,148.822
C09930=1237.256,-34.252,-38.731,-179.724,5.231,148.821
C09931=1237.251,-34.003,-38.744,-179.722,5.231,148.820
C09932=1237.246,-33.753,-38.757,-179.720,5.232,148.819
C09933=1237.240,-33.504,-38.770,-179.717,5.231,148.819
C09934=1237.236,-33.254,-38.784,-179.715,5.232,148.818
C09935=1237.230,-33.005,-38.797,-179.712,5.232,148.817
C09936=1237.226,-32.755,-38.810,-179.710,5.232,148.817
C09937=1237.220,-32.506,-38.824,-179.707,5.233,148.816
C09938=1237.216,-32.256,-38.837,-179.705,5.232,148.815
C09939=1237.210,-32.006,-38.850,-179.703,5.233,148.815
C09940=1237.206,-31.757,-38.864,-179.699,5.233,148.814
C09941=1237.200,-31.507,-38.877,-179.697,5.233,148.813
C09942=1237.195,-31.257,-38.890,-179.695,5.233,148.812
C09943=1237.190,-31.008,-38.904,-179.693,5.233,148.812
C09944=1237.185,-30.758,-38.917,-179.690,5.233,148.811
C09945=1237.180,-30.509,-38.931,-179.687,5.234,148.810
C09946=1237.175,-30.259,-38.944,-179.685,5.234,148.809
C09947=1237.169,-30.009,-38.957,-179.683,5.234,148.809
C09948=1237.165,-29.760,-38.971,-179.680,5.234,148.808
C09949=1237.159,-29.510,-38.984,-179.678,5.234,148.807
C09950=1237.155,-29.261,-38.997,-179.675,5.235,148.807
C09951=1237.149,-29.011,-39.011,-179.673,5.234,148.806
C09952=1237.144,-28.761,-39.025,-179.670,5.235,148.805
C09953=1237.139,-28.512,-39.037,-179.668,5.234,148.804
C09954=1237.134,-28.262,-39.052,-179.665,5.235,148.804
C09955=1237.129,-28.013,-39.064,-179.663,5.235,148.803
C09956=1237.124,-27.763,-39.079,-179.660,5.235,148.802
C09957=1237.119,-27.513,-39.092,-179.658,5.236,148.802
C09958=1237.114,-27.264,-39.105,-179.656,5.235,148.801
C09959=1237.109,-27.014,-39.119,-179.653,5.236,148.800
C09960=1237.104,-26.765,-39.132,-179.650,5.236,148.799
C09961=1237.099,-26.515,-39.146,-179.648,5.236,148.799
C09962=1237.094,-26.266,-39.159,-179.646,5.236,148.798
C09963=1237.089,-26.016,-39.173,-179.644,5.236,148.797
C09964=1237.084,-25.766,-39.187,-179.641,5.237,148.797
C09965=1237.078,-25.517,-39.200,-179.638,5.237,148.796
C09966=1237.073,-25.267,-39.214,-179.636,5.237,148.795
C09967=1237.068,-25.018,-39.227,-179.633,5.237,148.794
C09968=1237.063,-24.768,-39.241,-179.631,5.237,148.794
C09969=1237.058,-24.519,-39.254,-179.628,5.237,148.793
C09970=1237.053,-24.269,-39.268,-179.626,5.238,148.792
C09971=1237.048,-24.019,-39.282,-179.623,5.237,148.792
C09972=1237.043,-23.770,-39.295,-179.621,5.238,148.791
C09973=1237.038,-23.520,-39.309,-179.618,5.239,148.790
C09974=1237.033,-23.271,-39.323,-179.616,5.238,148.789
C09975=1237.027,-23.021,-39.336,-179.613,5.239,148.789
C09976=1237.023,-22.772,-39.350,-179.611,5.238,148.788
C09977=1237.018,-22.502,-39.365,-179.608,5.239,148.787
C09978=1237.012,-22.234,-39.380,-179.606,5.239,148.786
C09979=1237.006,-21.964,-39.395,-179.603,5.240,148.786
C09980=1237.001,-21.695,-39.410,-179.600,5.239,148.785
C09981=1236.996,-21.444,-39.423,-179.598,5.239,148.784
C09982=1236.991,-21.196,-39.437,-179.595,5.240,148.783
C09983=1236.986,-20.946,-39.451,-179.593,5.240,148.783
C09984=1236.980,-20.696,-39.464,-179.590,5.240,148.782
C09985=1236.976,-20.447,-39.478,-179.588,5.240,148.781
C09986=1236.971,-20.197,-39.492,-179.585,5.240,148.781
C09987=1236.965,-19.948,-39.506,-179.583,5.241,148.780
C09988=1236.960,-19.698,-39.519,-179.581,5.241,148.779
C09989=1236.956,-19.449,-39.533,-179.578,5.241,148.779
C09990=1236.950,-19.200,-39.547,-179.575,5.242,148.778
C09991=1236.945,-18.949,-39.561,-179.573,5.241,148.777
C09992=1236.940,-18.699,-39.575,-179.571,5.242,148.777
C09993=1236.934,-18.450,-39.589,-179.568,5.242,148.776
C09994=1236.930,-18.201,-39.602,-179.565,5.242,148.775
C09995=1236.925,-17.951,-39.617,-179.563,5.242,148.774
C09996=1236.919,-17.702,-39.630,-179.561,5.242,148.773
//INST
///DATE 2021/06/25 14:26
///ATTR SC,RW,RJ
////FRAME ROBOT
///GROUP1 RB1
NOP
MOVL C00000 V=800.0 PL=0
MOVL C00001 V=800.0 PL=0
MOVL C00002 V=800.0 PL=0
MOVL C00003 V=800.0 PL=0
MOVL C00004 V=800.0 PL=0
MOVL C00005 V=800.0 PL=0
MOVL C00006 V=800.0 PL=0
MOVL C00007 V=800.0 PL=0
MOVL C00008 V=800.0 PL=0
MOVL C00009 V=800.0 PL=0
MOVL C00010 V=800.0 PL=0
MOVL C00011 V=800.0 PL=0
MOVL C00012 V=800.0 PL=0
MOVL C00013 V=800.0 PL=0
MOVL C00014 V=800.0 PL=0
MOVL C00015 V=800.0 PL=0
MOVL C00016 V=800.0 PL=0
MOVL C00017 V=800.0 PL=0
MOVL C00018 V=800.0 PL=0
MOVL C00019 V=800.0 PL=0
MOVL C00020 V=800.0 PL=0
MOVL C00021 V=800.0 PL=0
MOVL C00022 V=800.0 PL=0
MOVL C00023 V=800.0 PL=0
MOVL C00024 V=800.0 PL=0
MOVL C00025 V=800.0 PL=0
MOVL C00026 V=800.0 PL=0
MOVL C00027 V=800.0 PL=0
MOVL C00028 V=800.0 PL=0
MOVL C00029 V=800.0 PL=0
MOVL C00030 V=800.0 PL=0
MOVL C00031 V=800.0 PL=0
MOVL C00032 V=800.0 PL=0
MOVL C00033 V=800.0 PL=0
MOVL C00034 V=800.0 PL=0
MOVL C00035 V=800.0 PL=0
MOVL C00036 V=800.0 PL=0
MOVL C00037 V=800.0 PL=0
MOVL C00038 V=800.0 PL=0
MOVL C00039 V=800.0 PL=0
MOVL C00040 V=800.0 PL=0
MOVL C00041 V=800.0 PL=0
MOVL C00042 V=800.0 PL=0
MOVL C00043 V=800.0 PL=0
MOVL C00044 V=800.0 PL=0
MOVL C00045 V=800.0 PL=0
MOVL C00046 V=800.0 PL=0
MOVL C00047 V=800.0 PL=0
MOVL C00048 V=800.0 PL=0
MOVL C00049 V=800.0 PL=0
MOVL C00050 V=800.0 PL=0
MOVL C00051 V=800.0 PL=0
MOVL C00052 V=800.0 PL=0
MOVL C00053 V=800.0 PL=0
MOVL C00054 V=800.0 PL=0
MOVL C00055 V=800.0 PL=0
MOVL C00056 V=800.0 PL=0
MOVL C00057 V=800.0 PL=0
MOVL C00058 V=800.0 PL=0
MOVL C00059 V=800.0 PL=0
MOVL C00060 V=800.0 PL=0
MOVL C00061 V=800.0 PL=0
MOVL C00062 V=800.0 PL=0
MOVL C00063 V=800.0 PL=0
MOVL C00064 V=800.0 PL=0
MOVL C00065 V=800.0 PL=0
MOVL C00066 V=800.0 PL=0
MOVL C00067 V=800.0 PL=0
MOVL C00068 V=800.0 PL=0
MOVL C00069 V=800.0 PL=0
MOVL C00070 V=800.0 PL=0
MOVL C00071 V=800.0 PL=0
MOVL C00072 V=800.0 PL=0
MOVL C00073 V=800.0 PL=0
MOVL C00074 V=800.0 PL=0
MOVL C00075 V=800.0 PL=0
MOVL C00076 V=800.0 PL=0
MOVL C00077 V=800.0 PL=0
MOVL C00078 V=800.0 PL=0
MOVL C00079 V=800.0 PL=0
MOVL C00080 V=800.0 PL=0
MOVL C00081 V=800.0 PL=0
MOVL C00082 V=800.0 PL=0
MOVL C00083 V=800.0 PL=0
MOVL C00084 V=800.0 PL=0
MOVL C00085 V=800.0 PL=0
MOVL C00086 V=800.0 PL=0
MOVL C00087 V=800.0 PL=0
MOVL C00088 V=800.0 PL=0
MOVL C00089 V=800.0 PL=0
MOVL C00090 V=800.0 PL=0
MOVL C00091 V=800.0 PL=0
MOVL C00092 V=800.0 PL=0
MOVL C00093 V=800.0 PL=0
MOVL C00094 V=800.0 PL=0
MOVL C00095 V=800.0 PL=0
MOVL C00096 V=800.0 PL=0
MOVL C00097 V=800.0 PL=0
MOVL C00098 V=800.0 PL=0
MOVL C00099 V=800.0 PL=0
MOVL C00100 V=800.0 PL=0
MOVL C00101 V=800.0 PL=0
MOVL C00102 V=800.0 PL=0
MOVL C00103 V=800.0 PL=0
MOVL C00104 V=800.0 PL=0
MOVL C00105 V=800.0 PL=0
MOVL C00106 V=800.0 PL=0
MOVL C00107 V=800.0 PL=0
MOVL C00108 V=800.0 PL=0
MOVL C00109 V=800.0 PL=0
MOVL C00110 V=800.0 PL=0
MOVL C00111 V=800.0 PL=0
MOVL C00112 V=800.0 PL=0
MOVL C00113 V=800.0 PL=0
MOVL C00114 V=800.0 PL=0
MOVL C00115 V=800.0 PL=0
MOVL C00116 V=800.0 PL=0
MOVL C00117 V=800.0 PL=0
MOVL C00118 V=800.0 PL=0
MOVL C00119 V=800.0 PL=0
MOVL C00120 V=800.0 PL=0
MOVL C00121 V=800.0 PL=0
MOVL C00122 V=800.0 PL=0
MOVL C00123 V=800.0 PL=0
MOVL C00124 V=800.0 PL=0
MOVL C00125 V=800.0 PL=0
MOVL C00126 V=800.0 PL=0
MOVL C00127 V=800.0 PL=0
MOVL C00128 V=800.0 PL=0
MOVL C00129 V=800.0 PL=0
MOVL C00130 V=800.0 PL=0
MOVL C00131 V=800.0 PL=0
MOVL C00132 V=800.0 PL=0
MOVL C00133 V=800.0 PL=0
MOVL C00134 V=800.0 PL=0
MOVL C00135 V=800.0 PL=0
MOVL C00136 V=800.0 PL=0
MOVL C00137 V=800.0 PL=0
MOVL C00138 V=800.0 PL=0
MOVL C00139 V=800.0 PL=0
MOVL C00140 V=800.0 PL=0
MOVL C00141 V=800.0 PL=0
MOVL C00142 V=800.0 PL=0
MOVL C00143 V=800.0 PL=0
MOVL C00144 V=800.0 PL=0
MOVL C00145 V=800.0 PL=0
MOVL C00146 V=800.0 PL=0
MOVL C00147 V=800.0 PL=0
MOVL C00148 V=800.0 PL=0
MOVL C00149 V=800.0 PL=0
MOVL C00150 V=800.0 PL=0
MOVL C00151 V=800.0 PL=0
MOVL C00152 V=800.0 PL=0
MOVL C00153 V=800.0 PL=0
MOVL C00154 V=800.0 PL=0
MOVL C00155 V=800.0 PL=0
MOVL C00156 V=800.0 PL=0
MOVL C00157 V=800.0 PL=0
MOVL C00158 V=800.0 PL=0
MOVL C00159 V=800.0 PL=0
MOVL C00160 V=800.0 PL=0
MOVL C00161 V=800.0 PL=0
MOVL C00162 V=800.0 PL=0
MOVL C00163 V=800.0 PL=0
MOVL C00164 V=800.0 PL=0
MOVL C00165 V=800.0 PL=0
MOVL C00166 V=800.0 PL=0
MOVL C00167 V=800.0 PL=0
MOVL C00168 V=800.0 PL=0
MOVL C00169 V=800.0 PL=0
MOVL C00170 V=800.0 PL=0
MOVL C00171 V=800.0 PL=0
MOVL C00172 V=800.0 PL=0
MOVL C00173 V=800.0 PL=0
MOVL C00174 V=800.0 PL=0
MOVL C00175 V=800.0 PL=0
MOVL C00176 V=800.0 PL=0
MOVL C00177 V=800.0 PL=0
MOVL C00178 V=800.0 PL=0
MOVL C00179 V=800.0 PL=0
MOVL C00180 V=800.0 PL=0
MOVL C00181 V=800.0 PL=0
MOVL C00182 V=800.0 PL=0
MOVL C00183 V=800.0 PL=0
MOVL C00184 V=800.0 PL=0
MOVL C00185 V=800.0 PL=0
MOVL C00186 V=800.0 PL=0
MOVL C00187 V=800.0 PL=0
MOVL C00188 V=800.0 PL=0
MOVL C00189 V=800.0 PL=0
MOVL C00190 V=800.0 PL=0
MOVL C00191 V=800.0 PL=0
MOVL C00192 V=800.0 PL=0
MOVL C00193 V=800.0 PL=0
MOVL C00194 V=800.0 PL=0
MOVL C00195 V=800.0 PL=0
MOVL C00196 V=800.0 PL=0
MOVL C00197 V=800.0 PL=0
MOVL C00198 V=800.0 PL=0
MOVL C00199 V=800.0 PL=0
MOVL C00200 V=800.0 PL=0
MOVL C00201 V=800.0 PL=0
MOVL C00202 V=800.0 PL=0
MOVL C00203 V=800.0 PL=0
MOVL C00204 V=800.0 PL=0
MOVL C00205 V=800.0 PL=0
MOVL C00206 V=800.0 PL=0
MOVL C00207 V=800.0 PL=0
MOVL C00208 V=800.0 PL=0
MOVL C00209 V=800.0 PL=0
MOVL C00210 V=800.0 PL=0
MOVL C00211 V=800.0 PL=0
MOVL C00212 V=800.0 PL=0
MOVL C00213 V=800.0 PL=0
MOVL C00214 V=800.0 PL=0
MOVL C00215 V=800.0 PL=0
MOVL C00216 V=800.0 PL=0
MOVL C00217 V=800.0 PL=0
MOVL C00218 V=800.0 PL=0
MOVL C00219 V=800.0 PL=0
MOVL C00220 V=800.0 PL=0
MOVL C00221 V=800.0 PL=0
MOVL C00222 V=800.0 PL=0
MOVL C00223 V=800.0 PL=0
MOVL C00224 V=800.0 PL=0
MOVL C00225 V=800.0 PL=0
MOVL C00226 V=800.0 PL=0
MOVL C00227 V=800.0 PL=0
MOVL C00228 V=800.0 PL=0
MOVL C00229 V=800.0 PL=0
MOVL C00230 V=800.0 PL=0
MOVL C00231 V=800.0 PL=0
MOVL C00232 V=800.0 PL=0
MOVL C00233 V=800.0 PL=0
MOVL C00234 V=800.0 PL=0
MOVL C00235 V=800.0 PL=0
MOVL C00236 V=800.0 PL=0
MOVL C00237 V=800.0 PL=0
MOVL C00238 V=800.0 PL=0
MOVL C00239 V=800.0 PL=0
MOVL C00240 V=800.0 PL=0
MOVL C00241 V=800.0 PL=0
MOVL C00242 V=800.0 PL=0
MOVL C00243 V=800.0 PL=0
MOVL C00244 V=800.0 PL=0
MOVL C00245 V=800.0 PL=0
MOVL C00246 V=800.0 PL=0
MOVL C00247 V=800.0 PL=0
MOVL C00248 V=800.0 PL=0
MOVL C00249 V=800.0 PL=0
MOVL C00250 V=800.0 PL=0
MOVL C00251 V=800.0 PL=0
MOVL C00252 V=800.0 PL=0
MOVL C00253 V=800.0 PL=0
MOVL C00254 V=800.0 PL=0
MOVL C00255 V=800.0 PL=0
MOVL C00256 V=800.0 PL=0
MOVL C00257 V=800.0 PL=0
MOVL C00258 V=800.0 PL=0
MOVL C00259 V=800.0 PL=0
MOVL C00260 V=800.0 PL=0
MOVL C00261 V=800.0 PL=0
MOVL C00262 V=800.0 PL=0
MOVL C00263 V=800.0 PL=0
MOVL C00264 V=800.0 PL=0
MOVL C00265 V=800.0 PL=0
MOVL C00266 V=800.0 PL=0
MOVL C00267 V=800.0 PL=0
MOVL C00268 V=800.0 PL=0
MOVL C00269 V=800.0 PL=0
MOVL C00270 V=800.0 PL=0
MOVL C00271 V=800.0 PL=0
MOVL C00272 V=800.0 PL=0
MOVL C00273 V=800.0 PL=0
MOVL C00274 V=800.0 PL=0
MOVL C00275 V=800.0 PL=0
MOVL C00276 V=800.0 PL=0
MOVL C00277 V=800.0 PL=0
MOVL C00278 V=800.0 PL=0
MOVL C00279 V=800.0 PL=0
MOVL C00280 V=800.0 PL=0
MOVL C00281 V=800.0 PL=0
MOVL C00282 V=800.0 PL=0
MOVL C00283 V=800.0 PL=0
MOVL C00284 V=800.0 PL=0
MOVL C00285 V=800.0 PL=0
MOVL C00286 V=800.0 PL=0
MOVL C00287 V=800.0 PL=0
MOVL C00288 V=800.0 PL=0
MOVL C00289 V=800.0 PL=0
MOVL C00290 V=800.0 PL=0
MOVL C00291 V=800.0 PL=0
MOVL C00292 V=800.0 PL=0
MOVL C00293 V=800.0 PL=0
MOVL C00294 V=800.0 PL=0
MOVL C00295 V=800.0 PL=0
MOVL C00296 V=800.0 PL=0
MOVL C00297 V=800.0 PL=0
MOVL C00298 V=800.0 PL=0
MOVL C00299 V=800.0 PL=0
MOVL C00300 V=800.0 PL=0
MOVL C00301 V=800.0 PL=0
MOVL C00302 V=800.0 PL=0
MOVL C00303 V=800.0 PL=0
MOVL C00304 V=800.0 PL=0
MOVL C00305 V=800.0 PL=0
MOVL C00306 V=800.0 PL=0
MOVL C00307 V=800.0 PL=0
MOVL C00308 V=800.0 PL=0
MOVL C00309 V=800.0 PL=0
MOVL C00310 V=800.0 PL=0
MOVL C00311 V=800.0 PL=0
MOVL C00312 V=800.0 PL=0
MOVL C00313 V=800.0 PL=0
MOVL C00314 V=800.0 PL=0
MOVL C00315 V=800.0 PL=0
MOVL C00316 V=800.0 PL=0
MOVL C00317 V=800.0 PL=0
MOVL C00318 V=800.0 PL=0
MOVL C00319 V=800.0 PL=0
MOVL C00320 V=800.0 PL=0
MOVL C00321 V=800.0 PL=0
MOVL C00322 V=800.0 PL=0
MOVL C00323 V=800.0 PL=0
MOVL C00324 V=800.0 PL=0
MOVL C00325 V=800.0 PL=0
MOVL C00326 V=800.0 PL=0
MOVL C00327 V=800.0 PL=0
MOVL C00328 V=800.0 PL=0
MOVL C00329 V=800.0 PL=0
MOVL C00330 V=800.0 PL=0
MOVL C00331 V=800.0 PL=0
MOVL C00332 V=800.0 PL=0
MOVL C00333 V=800.0 PL=0
MOVL C00334 V=800.0 PL=0
MOVL C00335 V=800.0 PL=0
MOVL C00336 V=800.0 PL=0
MOVL C00337 V=800.0 PL=0
MOVL C00338 V=800.0 PL=0
MOVL C00339 V=800.0 PL=0
MOVL C00340 V=800.0 PL=0
MOVL C00341 V=800.0 PL=0
MOVL C00342 V=800.0 PL=0
MOVL C00343 V=800.0 PL=0
MOVL C00344 V=800.0 PL=0
MOVL C00345 V=800.0 PL=0
MOVL C00346 V=800.0 PL=0
MOVL C00347 V=800.0 PL=0
MOVL C00348 V=800.0 PL=0
MOVL C00349 V=800.0 PL=0
MOVL C00350 V=800.0 PL=0
MOVL C00351 V=800.0 PL=0
MOVL C00352 V=800.0 PL=0
MOVL C00353 V=800.0 PL=0
MOVL C00354 V=800.0 PL=0
MOVL C00355 V=800.0 PL=0
MOVL C00356 V=800.0 PL=0
MOVL C00357 V=800.0 PL=0
MOVL C00358 V=800.0 PL=0
MOVL C00359 V=800.0 PL=0
MOVL C00360 V=800.0 PL=0
MOVL C00361 V=800.0 PL=0
MOVL C00362 V=800.0 PL=0
MOVL C00363 V=800.0 PL=0
MOVL C00364 V=800.0 PL=0
MOVL C00365 V=800.0 PL=0
MOVL C00366 V=800.0 PL=0
MOVL C00367 V=800.0 PL=0
MOVL C00368 V=800.0 PL=0
MOVL C00369 V=800.0 PL=0
MOVL C00370 V=800.0 PL=0
MOVL C00371 V=800.0 PL=0
MOVL C00372 V=800.0 PL=0
MOVL C00373 V=800.0 PL=0
MOVL C00374 V=800.0 PL=0
MOVL C00375 V=800.0 PL=0
MOVL C00376 V=800.0 PL=0
MOVL C00377 V=800.0 PL=0
MOVL C00378 V=800.0 PL=0
MOVL C00379 V=800.0 PL=0
MOVL C00380 V=800.0 PL=0
MOVL C00381 V=800.0 PL=0
MOVL C00382 V=800.0 PL=0
MOVL C00383 V=800.0 PL=0
MOVL C00384 V=800.0 PL=0
MOVL C00385 V=800.0 PL=0
MOVL C00386 V=800.0 PL=0
MOVL C00387 V=800.0 PL=0
MOVL C00388 V=800.0 PL=0
MOVL C00389 V=800.0 PL=0
MOVL C00390 V=800.0 PL=0
MOVL C00391 V=800.0 PL=0
MOVL C00392 V=800.0 PL=0
MOVL C00393 V=800.0 PL=0
MOVL C00394 V=800.0 PL=0
MOVL C00395 V=800.0 PL=0
MOVL C00396 V=800.0 PL=0
MOVL C00397 V=800.0 PL=0
MOVL C00398 V=800.0 PL=0
MOVL C00399 V=800.0 PL=0
MOVL C00400 V=800.0 PL=0
MOVL C00401 V=800.0 PL=0
MOVL C00402 V=800.0 PL=0
MOVL C00403 V=800.0 PL=0
MOVL C00404 V=800.0 PL=0
MOVL C00405 V=800.0 PL=0
MOVL C00406 V=800.0 PL=0
MOVL C00407 V=800.0 PL=0
MOVL C00408 V=800.0 PL=0
MOVL C00409 V=800.0 PL=0
MOVL C00410 V=800.0 PL=0
MOVL C00411 V=800.0 PL=0
MOVL C00412 V=800.0 PL=0
MOVL C00413 V=800.0 PL=0
MOVL C00414 V=800.0 PL=0
MOVL C00415 V=800.0 PL=0
MOVL C00416 V=800.0 PL=0
MOVL C00417 V=800.0 PL=0
MOVL C00418 V=800.0 PL=0
MOVL C00419 V=800.0 PL=0
MOVL C00420 V=800.0 PL=0
MOVL C00421 V=800.0 PL=0
MOVL C00422 V=800.0 PL=0
MOVL C00423 V=800.0 PL=0
MOVL C00424 V=800.0 PL=0
MOVL C00425 V=800.0 PL=0
MOVL C00426 V=800.0 PL=0
MOVL C00427 V=800.0 PL=0
MOVL C00428 V=800.0 PL=0
MOVL C00429 V=800.0 PL=0
MOVL C00430 V=800.0 PL=0
MOVL C00431 V=800.0 PL=0
MOVL C00432 V=800.0 PL=0
MOVL C00433 V=800.0 PL=0
MOVL C00434 V=800.0 PL=0
MOVL C00435 V=800.0 PL=0
MOVL C00436 V=800.0 PL=0
MOVL C00437 V=800.0 PL=0
MOVL C00438 V=800.0 PL=0
MOVL C00439 V=800.0 PL=0
MOVL C00440 V=800.0 PL=0
MOVL C00441 V=800.0 PL=0
MOVL C00442 V=800.0 PL=0
MOVL C00443 V=800.0 PL=0
MOVL C00444 V=800.0 PL=0
MOVL C00445 V=800.0 PL=0
MOVL C00446 V=800.0 PL=0
MOVL C00447 V=800.0 PL=0
MOVL C00448 V=800.0 PL=0
MOVL C00449 V=800.0 PL=0
MOVL C00450 V=800.0 PL=0
MOVL C00451 V=800.0 PL=0
MOVL C00452 V=800.0 PL=0
MOVL C00453 V=800.0 PL=0
MOVL C00454 V=800.0 PL=0
MOVL C00455 V=800.0 PL=0
MOVL C00456 V=800.0 PL=0
MOVL C00457 V=800.0 PL=0
MOVL C00458 V=800.0 PL=0
MOVL C00459 V=800.0 PL=0
MOVL C00460 V=800.0 PL=0
MOVL C00461 V=800.0 PL=0
MOVL C00462 V=800.0 PL=0
MOVL C00463 V=800.0 PL=0
MOVL C00464 V=800.0 PL=0
MOVL C00465 V=800.0 PL=0
MOVL C00466 V=800.0 PL=0
MOVL C00467 V=800.0 PL=0
MOVL C00468 V=800.0 PL=0
MOVL C00469 V=800.0 PL=0
MOVL C00470 V=800.0 PL=0
MOVL C00471 V=800.0 PL=0
MOVL C00472 V=800.0 PL=0
MOVL C00473 V=800.0 PL=0
MOVL C00474 V=800.0 PL=0
MOVL C00475 V=800.0 PL=0
MOVL C00476 V=800.0 PL=0
MOVL C00477 V=800.0 PL=0
MOVL C00478 V=800.0 PL=0
MOVL C00479 V=800.0 PL=0
MOVL C00480 V=800.0 PL=0
MOVL C00481 V=800.0 PL=0
MOVL C00482 V=800.0 PL=0
MOVL C00483 V=800.0 PL=0
MOVL C00484 V=800.0 PL=0
MOVL C00485 V=800.0 PL=0
MOVL C00486 V=800.0 PL=0
MOVL C00487 V=800.0 PL=0
MOVL C00488 V=800.0 PL=0
MOVL C00489 V=800.0 PL=0
MOVL C00490 V=800.0 PL=0
MOVL C00491 V=800.0 PL=0
MOVL C00492 V=800.0 PL=0
MOVL C00493 V=800.0 PL=0
MOVL C00494 V=800.0 PL=0
MOVL C00495 V=800.0 PL=0
MOVL C00496 V=800.0 PL=0
MOVL C00497 V=800.0 PL=0
MOVL C00498 V=800.0 PL=0
MOVL C00499 V=800.0 PL=0
MOVL C00500 V=800.0 PL=0
MOVL C00501 V=800.0 PL=0
MOVL C00502 V=800.0 PL=0
MOVL C00503 V=800.0 PL=0
MOVL C00504 V=800.0 PL=0
MOVL C00505 V=800.0 PL=0
MOVL C00506 V=800.0 PL=0
MOVL C00507 V=800.0 PL=0
MOVL C00508 V=800.0 PL=0
MOVL C00509 V=800.0 PL=0
MOVL C00510 V=800.0 PL=0
MOVL C00511 V=800.0 PL=0
MOVL C00512 V=800.0 PL=0
MOVL C00513 V=800.0 PL=0
MOVL C00514 V=800.0 PL=0
MOVL C00515 V=800.0 PL=0
MOVL C00516 V=800.0 PL=0
MOVL C00517 V=800.0 PL=0
MOVL C00518 V=800.0 PL=0
MOVL C00519 V=800.0 PL=0
MOVL C00520 V=800.0 PL=0
MOVL C00521 V=800.0 PL=0
MOVL C00522 V=800.0 PL=0
MOVL C00523 V=800.0 PL=0
MOVL C00524 V=800.0 PL=0
MOVL C00525 V=800.0 PL=0
MOVL C00526 V=800.0 PL=0
MOVL C00527 V=800.0 PL=0
MOVL C00528 V=800.0 PL=0
MOVL C00529 V=800.0 PL=0
MOVL C00530 V=800.0 PL=0
MOVL C00531 V=800.0 PL=0
MOVL C00532 V=800.0 PL=0
MOVL C00533 V=800.0 PL=0
MOVL C00534 V=800.0 PL=0
MOVL C00535 V=800.0 PL=0
MOVL C00536 V=800.0 PL=0
MOVL C00537 V=800.0 PL=0
MOVL C00538 V=800.0 PL=0
MOVL C00539 V=800.0 PL=0
MOVL C00540 V=800.0 PL=0
MOVL C00541 V=800.0 PL=0
MOVL C00542 V=800.0 PL=0
MOVL C00543 V=800.0 PL=0
MOVL C00544 V=800.0 PL=0
MOVL C00545 V=800.0 PL=0
MOVL C00546 V=800.0 PL=0
MOVL C00547 V=800.0 PL=0
MOVL C00548 V=800.0 PL=0
MOVL C00549 V=800.0 PL=0
MOVL C00550 V=800.0 PL=0
MOVL C00551 V=800.0 PL=0
MOVL C00552 V=800.0 PL=0
MOVL C00553 V=800.0 PL=0
MOVL C00554 V=800.0 PL=0
MOVL C00555 V=800.0 PL=0
MOVL C00556 V=800.0 PL=0
MOVL C00557 V=800.0 PL=0
MOVL C00558 V=800.0 PL=0
MOVL C00559 V=800.0 PL=0
MOVL C00560 V=800.0 PL=0
MOVL C00561 V=800.0 PL=0
MOVL C00562 V=800.0 PL=0
MOVL C00563 V=800.0 PL=0
MOVL C00564 V=800.0 PL=0
MOVL C00565 V=800.0 PL=0
MOVL C00566 V=800.0 PL=0
MOVL C00567 V=800.0 PL=0
MOVL C00568 V=800.0 PL=0
MOVL C00569 V=800.0 PL=0
MOVL C00570 V=800.0 PL=0
MOVL C00571 V=800.0 PL=0
MOVL C00572 V=800.0 PL=0
MOVL C00573 V=800.0 PL=0
MOVL C00574 V=800.0 PL=0
MOVL C00575 V=800.0 PL=0
MOVL C00576 V=800.0 PL=0
MOVL C00577 V=800.0 PL=0
MOVL C00578 V=800.0 PL=0
MOVL C00579 V=800.0 PL=0
MOVL C00580 V=800.0 PL=0
MOVL C00581 V=800.0 PL=0
MOVL C00582 V=800.0 PL=0
MOVL C00583 V=800.0 PL=0
MOVL C00584 V=800.0 PL=0
MOVL C00585 V=800.0 PL=0
MOVL C00586 V=800.0 PL=0
MOVL C00587 V=800.0 PL=0
MOVL C00588 V=800.0 PL=0
MOVL C00589 V=800.0 PL=0
MOVL C00590 V=800.0 PL=0
MOVL C00591 V=800.0 PL=0
MOVL C00592 V=800.0 PL=0
MOVL C00593 V=800.0 PL=0
MOVL C00594 V=800.0 PL=0
MOVL C00595 V=800.0 PL=0
MOVL C00596 V=800.0 PL=0
MOVL C00597 V=800.0 PL=0
MOVL C00598 V=800.0 PL=0
MOVL C00599 V=800.0 PL=0
MOVL C00600 V=800.0 PL=0
MOVL C00601 V=800.0 PL=0
MOVL C00602 V=800.0 PL=0
MOVL C00603 V=800.0 PL=0
MOVL C00604 V=800.0 PL=0
MOVL C00605 V=800.0 PL=0
MOVL C00606 V=800.0 PL=0
MOVL C00607 V=800.0 PL=0
MOVL C00608 V=800.0 PL=0
MOVL C00609 V=800.0 PL=0
MOVL C00610 V=800.0 PL=0
MOVL C00611 V=800.0 PL=0
MOVL C00612 V=800.0 PL=0
MOVL C00613 V=800.0 PL=0
MOVL C00614 V=800.0 PL=0
MOVL C00615 V=800.0 PL=0
MOVL C00616 V=800.0 PL=0
MOVL C00617 V=800.0 PL=0
MOVL C00618 V=800.0 PL=0
MOVL C00619 V=800.0 PL=0
MOVL C00620 V=800.0 PL=0
MOVL C00621 V=800.0 PL=0
MOVL C00622 V=800.0 PL=0
MOVL C00623 V=800.0 PL=0
MOVL C00624 V=800.0 PL=0
MOVL C00625 V=800.0 PL=0
MOVL C00626 V=800.0 PL=0
MOVL C00627 V=800.0 PL=0
MOVL C00628 V=800.0 PL=0
MOVL C00629 V=800.0 PL=0
MOVL C00630 V=800.0 PL=0
MOVL C00631 V=800.0 PL=0
MOVL C00632 V=800.0 PL=0
MOVL C00633 V=800.0 PL=0
MOVL C00634 V=800.0 PL=0
MOVL C00635 V=800.0 PL=0
MOVL C00636 V=800.0 PL=0
MOVL C00637 V=800.0 PL=0
MOVL C00638 V=800.0 PL=0
MOVL C00639 V=800.0 PL=0
MOVL C00640 V=800.0 PL=0
MOVL C00641 V=800.0 PL=0
MOVL C00642 V=800.0 PL=0
MOVL C00643 V=800.0 PL=0
MOVL C00644 V=800.0 PL=0
MOVL C00645 V=800.0 PL=0
MOVL C00646 V=800.0 PL=0
MOVL C00647 V=800.0 PL=0
MOVL C00648 V=800.0 PL=0
MOVL C00649 V=800.0 PL=0
MOVL C00650 V=800.0 PL=0
MOVL C00651 V=800.0 PL=0
MOVL C00652 V=800.0 PL=0
MOVL C00653 V=800.0 PL=0
MOVL C00654 V=800.0 PL=0
MOVL C00655 V=800.0 PL=0
MOVL C00656 V=800.0 PL=0
MOVL C00657 V=800.0 PL=0
MOVL C00658 V=800.0 PL=0
MOVL C00659 V=800.0 PL=0
MOVL C00660 V=800.0 PL=0
MOVL C00661 V=800.0 PL=0
MOVL C00662 V=800.0 PL=0
MOVL C00663 V=800.0 PL=0
MOVL C00664 V=800.0 PL=0
MOVL C00665 V=800.0 PL=0
MOVL C00666 V=800.0 PL=0
MOVL C00667 V=800.0 PL=0
MOVL C00668 V=800.0 PL=0
MOVL C00669 V=800.0 PL=0
MOVL C00670 V=800.0 PL=0
MOVL C00671 V=800.0 PL=0
MOVL C00672 V=800.0 PL=0
MOVL C00673 V=800.0 PL=0
MOVL C00674 V=800.0 PL=0
MOVL C00675 V=800.0 PL=0
MOVL C00676 V=800.0 PL=0
MOVL C00677 V=800.0 PL=0
MOVL C00678 V=800.0 PL=0
MOVL C00679 V=800.0 PL=0
MOVL C00680 V=800.0 PL=0
MOVL C00681 V=800.0 PL=0
MOVL C00682 V=800.0 PL=0
MOVL C00683 V=800.0 PL=0
MOVL C00684 V=800.0 PL=0
MOVL C00685 V=800.0 PL=0
MOVL C00686 V=800.0 PL=0
MOVL C00687 V=800.0 PL=0
MOVL C00688 V=800.0 PL=0
MOVL C00689 V=800.0 PL=0
MOVL C00690 V=800.0 PL=0
MOVL C00691 V=800.0 PL=0
MOVL C00692 V=800.0 PL=0
MOVL C00693 V=800.0 PL=0
MOVL C00694 V=800.0 PL=0
MOVL C00695 V=800.0 PL=0
MOVL C00696 V=800.0 PL=0
MOVL C00697 V=800.0 PL=0
MOVL C00698 V=800.0 PL=0
MOVL C00699 V=800.0 PL=0
MOVL C00700 V=800.0 PL=0
MOVL C00701 V=800.0 PL=0
MOVL C00702 V=800.0 PL=0
MOVL C00703 V=800.0 PL=0
MOVL C00704 V=800.0 PL=0
MOVL C00705 V=800.0 PL=0
MOVL C00706 V=800.0 PL=0
MOVL C00707 V=800.0 PL=0
MOVL C00708 V=800.0 PL=0
MOVL C00709 V=800.0 PL=0
MOVL C00710 V=800.0 PL=0
MOVL C00711 V=800.0 PL=0
MOVL C00712 V=800.0 PL=0
MOVL C00713 V=800.0 PL=0
MOVL C00714 V=800.0 PL=0
MOVL C00715 V=800.0 PL=0
MOVL C00716 V=800.0 PL=0
MOVL C00717 V=800.0 PL=0
MOVL C00718 V=800.0 PL=0
MOVL C00719 V=800.0 PL=0
MOVL C00720 V=800.0 PL=0
MOVL C00721 V=800.0 PL=0
MOVL C00722 V=800.0 PL=0
MOVL C00723 V=800.0 PL=0
MOVL C00724 V=800.0 PL=0
MOVL C00725 V=800.0 PL=0
MOVL C00726 V=800.0 PL=0
MOVL C00727 V=800.0 PL=0
MOVL C00728 V=800.0 PL=0
MOVL C00729 V=800.0 PL=0
MOVL C00730 V=800.0 PL=0
MOVL C00731 V=800.0 PL=0
MOVL C00732 V=800.0 PL=0
MOVL C00733 V=800.0 PL=0
MOVL C00734 V=800.0 PL=0
MOVL C00735 V=800.0 PL=0
MOVL C00736 V=800.0 PL=0
MOVL C00737 V=800.0 PL=0
MOVL C00738 V=800.0 PL=0
MOVL C00739 V=800.0 PL=0
MOVL C00740 V=800.0 PL=0
MOVL C00741 V=800.0 PL=0
MOVL C00742 V=800.0 PL=0
MOVL C00743 V=800.0 PL=0
MOVL C00744 V=800.0 PL=0
MOVL C00745 V=800.0 PL=0
MOVL C00746 V=800.0 PL=0
MOVL C00747 V=800.0 PL=0
MOVL C00748 V=800.0 PL=0
MOVL C00749 V=800.0 PL=0
MOVL C00750 V=800.0 PL=0
MOVL C00751 V=800.0 PL=0
MOVL C00752 V=800.0 PL=0
MOVL C00753 V=800.0 PL=0
MOVL C00754 V=800.0 PL=0
MOVL C00755 V=800.0 PL=0
MOVL C00756 V=800.0 PL=0
MOVL C00757 V=800.0 PL=0
MOVL C00758 V=800.0 PL=0
MOVL C00759 V=800.0 PL=0
MOVL C00760 V=800.0 PL=0
MOVL C00761 V=800.0 PL=0
MOVL C00762 V=800.0 PL=0
MOVL C00763 V=800.0 PL=0
MOVL C00764 V=800.0 PL=0
MOVL C00765 V=800.0 PL=0
MOVL C00766 V=800.0 PL=0
MOVL C00767 V=800.0 PL=0
MOVL C00768 V=800.0 PL=0
MOVL C00769 V=800.0 PL=0
MOVL C00770 V=800.0 PL=0
MOVL C00771 V=800.0 PL=0
MOVL C00772 V=800.0 PL=0
MOVL C00773 V=800.0 PL=0
MOVL C00774 V=800.0 PL=0
MOVL C00775 V=800.0 PL=0
MOVL C00776 V=800.0 PL=0
MOVL C00777 V=800.0 PL=0
MOVL C00778 V=800.0 PL=0
MOVL C00779 V=800.0 PL=0
MOVL C00780 V=800.0 PL=0
MOVL C00781 V=800.0 PL=0
MOVL C00782 V=800.0 PL=0
MOVL C00783 V=800.0 PL=0
MOVL C00784 V=800.0 PL=0
MOVL C00785 V=800.0 PL=0
MOVL C00786 V=800.0 PL=0
MOVL C00787 V=800.0 PL=0
MOVL C00788 V=800.0 PL=0
MOVL C00789 V=800.0 PL=0
MOVL C00790 V=800.0 PL=0
MOVL C00791 V=800.0 PL=0
MOVL C00792 V=800.0 PL=0
MOVL C00793 V=800.0 PL=0
MOVL C00794 V=800.0 PL=0
MOVL C00795 V=800.0 PL=0
MOVL C00796 V=800.0 PL=0
MOVL C00797 V=800.0 PL=0
MOVL C00798 V=800.0 PL=0
MOVL C00799 V=800.0 PL=0
MOVL C00800 V=800.0 PL=0
MOVL C00801 V=800.0 PL=0
MOVL C00802 V=800.0 PL=0
MOVL C00803 V=800.0 PL=0
MOVL C00804 V=800.0 PL=0
MOVL C00805 V=800.0 PL=0
MOVL C00806 V=800.0 PL=0
MOVL C00807 V=800.0 PL=0
MOVL C00808 V=800.0 PL=0
MOVL C00809 V=800.0 PL=0
MOVL C00810 V=800.0 PL=0
MOVL C00811 V=800.0 PL=0
MOVL C00812 V=800.0 PL=0
MOVL C00813 V=800.0 PL=0
MOVL C00814 V=800.0 PL=0
MOVL C00815 V=800.0 PL=0
MOVL C00816 V=800.0 PL=0
MOVL C00817 V=800.0 PL=0
MOVL C00818 V=800.0 PL=0
MOVL C00819 V=800.0 PL=0
MOVL C00820 V=800.0 PL=0
MOVL C00821 V=800.0 PL=0
MOVL C00822 V=800.0 PL=0
MOVL C00823 V=800.0 PL=0
MOVL C00824 V=800.0 PL=0
MOVL C00825 V=800.0 PL=0
MOVL C00826 V=800.0 PL=0
MOVL C00827 V=800.0 PL=0
MOVL C00828 V=800.0 PL=0
MOVL C00829 V=800.0 PL=0
MOVL C00830 V=800.0 PL=0
MOVL C00831 V=800.0 PL=0
MOVL C00832 V=800.0 PL=0
MOVL C00833 V=800.0 PL=0
MOVL C00834 V=800.0 PL=0
MOVL C00835 V=800.0 PL=0
MOVL C00836 V=800.0 PL=0
MOVL C00837 V=800.0 PL=0
MOVL C00838 V=800.0 PL=0
MOVL C00839 V=800.0 PL=0
MOVL C00840 V=800.0 PL=0
MOVL C00841 V=800.0 PL=0
MOVL C00842 V=800.0 PL=0
MOVL C00843 V=800.0 PL=0
MOVL C00844 V=800.0 PL=0
MOVL C00845 V=800.0 PL=0
MOVL C00846 V=800.0 PL=0
MOVL C00847 V=800.0 PL=0
MOVL C00848 V=800.0 PL=0
MOVL C00849 V=800.0 PL=0
MOVL C00850 V=800.0 PL=0
MOVL C00851 V=800.0 PL=0
MOVL C00852 V=800.0 PL=0
MOVL C00853 V=800.0 PL=0
MOVL C00854 V=800.0 PL=0
MOVL C00855 V=800.0 PL=0
MOVL C00856 V=800.0 PL=0
MOVL C00857 V=800.0 PL=0
MOVL C00858 V=800.0 PL=0
MOVL C00859 V=800.0 PL=0
MOVL C00860 V=800.0 PL=0
MOVL C00861 V=800.0 PL=0
MOVL C00862 V=800.0 PL=0
MOVL C00863 V=800.0 PL=0
MOVL C00864 V=800.0 PL=0
MOVL C00865 V=800.0 PL=0
MOVL C00866 V=800.0 PL=0
MOVL C00867 V=800.0 PL=0
MOVL C00868 V=800.0 PL=0
MOVL C00869 V=800.0 PL=0
MOVL C00870 V=800.0 PL=0
MOVL C00871 V=800.0 PL=0
MOVL C00872 V=800.0 PL=0
MOVL C00873 V=800.0 PL=0
MOVL C00874 V=800.0 PL=0
MOVL C00875 V=800.0 PL=0
MOVL C00876 V=800.0 PL=0
MOVL C00877 V=800.0 PL=0
MOVL C00878 V=800.0 PL=0
MOVL C00879 V=800.0 PL=0
MOVL C00880 V=800.0 PL=0
MOVL C00881 V=800.0 PL=0
MOVL C00882 V=800.0 PL=0
MOVL C00883 V=800.0 PL=0
MOVL C00884 V=800.0 PL=0
MOVL C00885 V=800.0 PL=0
MOVL C00886 V=800.0 PL=0
MOVL C00887 V=800.0 PL=0
MOVL C00888 V=800.0 PL=0
MOVL C00889 V=800.0 PL=0
MOVL C00890 V=800.0 PL=0
MOVL C00891 V=800.0 PL=0
MOVL C00892 V=800.0 PL=0
MOVL C00893 V=800.0 PL=0
MOVL C00894 V=800.0 PL=0
MOVL C00895 V=800.0 PL=0
MOVL C00896 V=800.0 PL=0
MOVL C00897 V=800.0 PL=0
MOVL C00898 V=800.0 PL=0
MOVL C00899 V=800.0 PL=0
MOVL C00900 V=800.0 PL=0
MOVL C00901 V=800.0 PL=0
MOVL C00902 V=800.0 PL=0
MOVL C00903 V=800.0 PL=0
MOVL C00904 V=800.0 PL=0
MOVL C00905 V=800.0 PL=0
MOVL C00906 V=800.0 PL=0
MOVL C00907 V=800.0 PL=0
MOVL C00908 V=800.0 PL=0
MOVL C00909 V=800.0 PL=0
MOVL C00910 V=800.0 PL=0
MOVL C00911 V=800.0 PL=0
MOVL C00912 V=800.0 PL=0
MOVL C00913 V=800.0 PL=0
MOVL C00914 V=800.0 PL=0
MOVL C00915 V=800.0 PL=0
MOVL C00916 V=800.0 PL=0
MOVL C00917 V=800.0 PL=0
MOVL C00918 V=800.0 PL=0
MOVL C00919 V=800.0 PL=0
MOVL C00920 V=800.0 PL=0
MOVL C00921 V=800.0 PL=0
MOVL C00922 V=800.0 PL=0
MOVL C00923 V=800.0 PL=0
MOVL C00924 V=800.0 PL=0
MOVL C00925 V=800.0 PL=0
MOVL C00926 V=800.0 PL=0
MOVL C00927 V=800.0 PL=0
MOVL C00928 V=800.0 PL=0
MOVL C00929 V=800.0 PL=0
MOVL C00930 V=800.0 PL=0
MOVL C00931 V=800.0 PL=0
MOVL C00932 V=800.0 PL=0
MOVL C00933 V=800.0 PL=0
MOVL C00934 V=800.0 PL=0
MOVL C00935 V=800.0 PL=0
MOVL C00936 V=800.0 PL=0
MOVL C00937 V=800.0 PL=0
MOVL C00938 V=800.0 PL=0
MOVL C00939 V=800.0 PL=0
MOVL C00940 V=800.0 PL=0
MOVL C00941 V=800.0 PL=0
MOVL C00942 V=800.0 PL=0
MOVL C00943 V=800.0 PL=0
MOVL C00944 V=800.0 PL=0
MOVL C00945 V=800.0 PL=0
MOVL C00946 V=800.0 PL=0
MOVL C00947 V=800.0 PL=0
MOVL C00948 V=800.0 PL=0
MOVL C00949 V=800.0 PL=0
MOVL C00950 V=800.0 PL=0
MOVL C00951 V=800.0 PL=0
MOVL C00952 V=800.0 PL=0
MOVL C00953 V=800.0 PL=0
MOVL C00954 V=800.0 PL=0
MOVL C00955 V=800.0 PL=0
MOVL C00956 V=800.0 PL=0
MOVL C00957 V=800.0 PL=0
MOVL C00958 V=800.0 PL=0
MOVL C00959 V=800.0 PL=0
MOVL C00960 V=800.0 PL=0
MOVL C00961 V=800.0 PL=0
MOVL C00962 V=800.0 PL=0
MOVL C00963 V=800.0 PL=0
MOVL C00964 V=800.0 PL=0
MOVL C00965 V=800.0 PL=0
MOVL C00966 V=800.0 PL=0
MOVL C00967 V=800.0 PL=0
MOVL C00968 V=800.0 PL=0
MOVL C00969 V=800.0 PL=0
MOVL C00970 V=800.0 PL=0
MOVL C00971 V=800.0 PL=0
MOVL C00972 V=800.0 PL=0
MOVL C00973 V=800.0 PL=0
MOVL C00974 V=800.0 PL=0
MOVL C00975 V=800.0 PL=0
MOVL C00976 V=800.0 PL=0
MOVL C00977 V=800.0 PL=0
MOVL C00978 V=800.0 PL=0
MOVL C00979 V=800.0 PL=0
MOVL C00980 V=800.0 PL=0
MOVL C00981 V=800.0 PL=0
MOVL C00982 V=800.0 PL=0
MOVL C00983 V=800.0 PL=0
MOVL C00984 V=800.0 PL=0
MOVL C00985 V=800.0 PL=0
MOVL C00986 V=800.0 PL=0
MOVL C00987 V=800.0 PL=0
MOVL C00988 V=800.0 PL=0
MOVL C00989 V=800.0 PL=0
MOVL C00990 V=800.0 PL=0
MOVL C00991 V=800.0 PL=0
MOVL C00992 V=800.0 PL=0
MOVL C00993 V=800.0 PL=0
MOVL C00994 V=800.0 PL=0
MOVL C00995 V=800.0 PL=0
MOVL C00996 V=800.0 PL=0
MOVL C00997 V=800.0 PL=0
MOVL C00998 V=800.0 PL=0
MOVL C00999 V=800.0 PL=0
MOVL C01000 V=800.0 PL=0
MOVL C01001 V=800.0 PL=0
MOVL C01002 V=800.0 PL=0
MOVL C01003 V=800.0 PL=0
MOVL C01004 V=800.0 PL=0
MOVL C01005 V=800.0 PL=0
MOVL C01006 V=800.0 PL=0
MOVL C01007 V=800.0 PL=0
MOVL C01008 V=800.0 PL=0
MOVL C01009 V=800.0 PL=0
MOVL C01010 V=800.0 PL=0
MOVL C01011 V=800.0 PL=0
MOVL C01012 V=800.0 PL=0
MOVL C01013 V=800.0 PL=0
MOVL C01014 V=800.0 PL=0
MOVL C01015 V=800.0 PL=0
MOVL C01016 V=800.0 PL=0
MOVL C01017 V=800.0 PL=0
MOVL C01018 V=800.0 PL=0
MOVL C01019 V=800.0 PL=0
MOVL C01020 V=800.0 PL=0
MOVL C01021 V=800.0 PL=0
MOVL C01022 V=800.0 PL=0
MOVL C01023 V=800.0 PL=0
MOVL C01024 V=800.0 PL=0
MOVL C01025 V=800.0 PL=0
MOVL C01026 V=800.0 PL=0
MOVL C01027 V=800.0 PL=0
MOVL C01028 V=800.0 PL=0
MOVL C01029 V=800.0 PL=0
MOVL C01030 V=800.0 PL=0
MOVL C01031 V=800.0 PL=0
MOVL C01032 V=800.0 PL=0
MOVL C01033 V=800.0 PL=0
MOVL C01034 V=800.0 PL=0
MOVL C01035 V=800.0 PL=0
MOVL C01036 V=800.0 PL=0
MOVL C01037 V=800.0 PL=0
MOVL C01038 V=800.0 PL=0
MOVL C01039 V=800.0 PL=0
MOVL C01040 V=800.0 PL=0
MOVL C01041 V=800.0 PL=0
MOVL C01042 V=800.0 PL=0
MOVL C01043 V=800.0 PL=0
MOVL C01044 V=800.0 PL=0
MOVL C01045 V=800.0 PL=0
MOVL C01046 V=800.0 PL=0
MOVL C01047 V=800.0 PL=0
MOVL C01048 V=800.0 PL=0
MOVL C01049 V=800.0 PL=0
MOVL C01050 V=800.0 PL=0
MOVL C01051 V=800.0 PL=0
MOVL C01052 V=800.0 PL=0
MOVL C01053 V=800.0 PL=0
MOVL C01054 V=800.0 PL=0
MOVL C01055 V=800.0 PL=0
MOVL C01056 V=800.0 PL=0
MOVL C01057 V=800.0 PL=0
MOVL C01058 V=800.0 PL=0
MOVL C01059 V=800.0 PL=0
MOVL C01060 V=800.0 PL=0
MOVL C01061 V=800.0 PL=0
MOVL C01062 V=800.0 PL=0
MOVL C01063 V=800.0 PL=0
MOVL C01064 V=800.0 PL=0
MOVL C01065 V=800.0 PL=0
MOVL C01066 V=800.0 PL=0
MOVL C01067 V=800.0 PL=0
MOVL C01068 V=800.0 PL=0
MOVL C01069 V=800.0 PL=0
MOVL C01070 V=800.0 PL=0
MOVL C01071 V=800.0 PL=0
MOVL C01072 V=800.0 PL=0
MOVL C01073 V=800.0 PL=0
MOVL C01074 V=800.0 PL=0
MOVL C01075 V=800.0 PL=0
MOVL C01076 V=800.0 PL=0
MOVL C01077 V=800.0 PL=0
MOVL C01078 V=800.0 PL=0
MOVL C01079 V=800.0 PL=0
MOVL C01080 V=800.0 PL=0
MOVL C01081 V=800.0 PL=0
MOVL C01082 V=800.0 PL=0
MOVL C01083 V=800.0 PL=0
MOVL C01084 V=800.0 PL=0
MOVL C01085 V=800.0 PL=0
MOVL C01086 V=800.0 PL=0
MOVL C01087 V=800.0 PL=0
MOVL C01088 V=800.0 PL=0
MOVL C01089 V=800.0 PL=0
MOVL C01090 V=800.0 PL=0
MOVL C01091 V=800.0 PL=0
MOVL C01092 V=800.0 PL=0
MOVL C01093 V=800.0 PL=0
MOVL C01094 V=800.0 PL=0
MOVL C01095 V=800.0 PL=0
MOVL C01096 V=800.0 PL=0
MOVL C01097 V=800.0 PL=0
MOVL C01098 V=800.0 PL=0
MOVL C01099 V=800.0 PL=0
MOVL C01100 V=800.0 PL=0
MOVL C01101 V=800.0 PL=0
MOVL C01102 V=800.0 PL=0
MOVL C01103 V=800.0 PL=0
MOVL C01104 V=800.0 PL=0
MOVL C01105 V=800.0 PL=0
MOVL C01106 V=800.0 PL=0
MOVL C01107 V=800.0 PL=0
MOVL C01108 V=800.0 PL=0
MOVL C01109 V=800.0 PL=0
MOVL C01110 V=800.0 PL=0
MOVL C01111 V=800.0 PL=0
MOVL C01112 V=800.0 PL=0
MOVL C01113 V=800.0 PL=0
MOVL C01114 V=800.0 PL=0
MOVL C01115 V=800.0 PL=0
MOVL C01116 V=800.0 PL=0
MOVL C01117 V=800.0 PL=0
MOVL C01118 V=800.0 PL=0
MOVL C01119 V=800.0 PL=0
MOVL C01120 V=800.0 PL=0
MOVL C01121 V=800.0 PL=0
MOVL C01122 V=800.0 PL=0
MOVL C01123 V=800.0 PL=0
MOVL C01124 V=800.0 PL=0
MOVL C01125 V=800.0 PL=0
MOVL C01126 V=800.0 PL=0
MOVL C01127 V=800.0 PL=0
MOVL C01128 V=800.0 PL=0
MOVL C01129 V=800.0 PL=0
MOVL C01130 V=800.0 PL=0
MOVL C01131 V=800.0 PL=0
MOVL C01132 V=800.0 PL=0
MOVL C01133 V=800.0 PL=0
MOVL C01134 V=800.0 PL=0
MOVL C01135 V=800.0 PL=0
MOVL C01136 V=800.0 PL=0
MOVL C01137 V=800.0 PL=0
MOVL C01138 V=800.0 PL=0
MOVL C01139 V=800.0 PL=0
MOVL C01140 V=800.0 PL=0
MOVL C01141 V=800.0 PL=0
MOVL C01142 V=800.0 PL=0
MOVL C01143 V=800.0 PL=0
MOVL C01144 V=800.0 PL=0
MOVL C01145 V=800.0 PL=0
MOVL C01146 V=800.0 PL=0
MOVL C01147 V=800.0 PL=0
MOVL C01148 V=800.0 PL=0
MOVL C01149 V=800.0 PL=0
MOVL C01150 V=800.0 PL=0
MOVL C01151 V=800.0 PL=0
MOVL C01152 V=800.0 PL=0
MOVL C01153 V=800.0 PL=0
MOVL C01154 V=800.0 PL=0
MOVL C01155 V=800.0 PL=0
MOVL C01156 V=800.0 PL=0
MOVL C01157 V=800.0 PL=0
MOVL C01158 V=800.0 PL=0
MOVL C01159 V=800.0 PL=0
MOVL C01160 V=800.0 PL=0
MOVL C01161 V=800.0 PL=0
MOVL C01162 V=800.0 PL=0
MOVL C01163 V=800.0 PL=0
MOVL C01164 V=800.0 PL=0
MOVL C01165 V=800.0 PL=0
MOVL C01166 V=800.0 PL=0
MOVL C01167 V=800.0 PL=0
MOVL C01168 V=800.0 PL=0
MOVL C01169 V=800.0 PL=0
MOVL C01170 V=800.0 PL=0
MOVL C01171 V=800.0 PL=0
MOVL C01172 V=800.0 PL=0
MOVL C01173 V=800.0 PL=0
MOVL C01174 V=800.0 PL=0
MOVL C01175 V=800.0 PL=0
MOVL C01176 V=800.0 PL=0
MOVL C01177 V=800.0 PL=0
MOVL C01178 V=800.0 PL=0
MOVL C01179 V=800.0 PL=0
MOVL C01180 V=800.0 PL=0
MOVL C01181 V=800.0 PL=0
MOVL C01182 V=800.0 PL=0
MOVL C01183 V=800.0 PL=0
MOVL C01184 V=800.0 PL=0
MOVL C01185 V=800.0 PL=0
MOVL C01186 V=800.0 PL=0
MOVL C01187 V=800.0 PL=0
MOVL C01188 V=800.0 PL=0
MOVL C01189 V=800.0 PL=0
MOVL C01190 V=800.0 PL=0
MOVL C01191 V=800.0 PL=0
MOVL C01192 V=800.0 PL=0
MOVL C01193 V=800.0 PL=0
MOVL C01194 V=800.0 PL=0
MOVL C01195 V=800.0 PL=0
MOVL C01196 V=800.0 PL=0
MOVL C01197 V=800.0 PL=0
MOVL C01198 V=800.0 PL=0
MOVL C01199 V=800.0 PL=0
MOVL C01200 V=800.0 PL=0
MOVL C01201 V=800.0 PL=0
MOVL C01202 V=800.0 PL=0
MOVL C01203 V=800.0 PL=0
MOVL C01204 V=800.0 PL=0
MOVL C01205 V=800.0 PL=0
MOVL C01206 V=800.0 PL=0
MOVL C01207 V=800.0 PL=0
MOVL C01208 V=800.0 PL=0
MOVL C01209 V=800.0 PL=0
MOVL C01210 V=800.0 PL=0
MOVL C01211 V=800.0 PL=0
MOVL C01212 V=800.0 PL=0
MOVL C01213 V=800.0 PL=0
MOVL C01214 V=800.0 PL=0
MOVL C01215 V=800.0 PL=0
MOVL C01216 V=800.0 PL=0
MOVL C01217 V=800.0 PL=0
MOVL C01218 V=800.0 PL=0
MOVL C01219 V=800.0 PL=0
MOVL C01220 V=800.0 PL=0
MOVL C01221 V=800.0 PL=0
MOVL C01222 V=800.0 PL=0
MOVL C01223 V=800.0 PL=0
MOVL C01224 V=800.0 PL=0
MOVL C01225 V=800.0 PL=0
MOVL C01226 V=800.0 PL=0
MOVL C01227 V=800.0 PL=0
MOVL C01228 V=800.0 PL=0
MOVL C01229 V=800.0 PL=0
MOVL C01230 V=800.0 PL=0
MOVL C01231 V=800.0 PL=0
MOVL C01232 V=800.0 PL=0
MOVL C01233 V=800.0 PL=0
MOVL C01234 V=800.0 PL=0
MOVL C01235 V=800.0 PL=0
MOVL C01236 V=800.0 PL=0
MOVL C01237 V=800.0 PL=0
MOVL C01238 V=800.0 PL=0
MOVL C01239 V=800.0 PL=0
MOVL C01240 V=800.0 PL=0
MOVL C01241 V=800.0 PL=0
MOVL C01242 V=800.0 PL=0
MOVL C01243 V=800.0 PL=0
MOVL C01244 V=800.0 PL=0
MOVL C01245 V=800.0 PL=0
MOVL C01246 V=800.0 PL=0
MOVL C01247 V=800.0 PL=0
MOVL C01248 V=800.0 PL=0
MOVL C01249 V=800.0 PL=0
MOVL C01250 V=800.0 PL=0
MOVL C01251 V=800.0 PL=0
MOVL C01252 V=800.0 PL=0
MOVL C01253 V=800.0 PL=0
MOVL C01254 V=800.0 PL=0
MOVL C01255 V=800.0 PL=0
MOVL C01256 V=800.0 PL=0
MOVL C01257 V=800.0 PL=0
MOVL C01258 V=800.0 PL=0
MOVL C01259 V=800.0 PL=0
MOVL C01260 V=800.0 PL=0
MOVL C01261 V=800.0 PL=0
MOVL C01262 V=800.0 PL=0
MOVL C01263 V=800.0 PL=0
MOVL C01264 V=800.0 PL=0
MOVL C01265 V=800.0 PL=0
MOVL C01266 V=800.0 PL=0
MOVL C01267 V=800.0 PL=0
MOVL C01268 V=800.0 PL=0
MOVL C01269 V=800.0 PL=0
MOVL C01270 V=800.0 PL=0
MOVL C01271 V=800.0 PL=0
MOVL C01272 V=800.0 PL=0
MOVL C01273 V=800.0 PL=0
MOVL C01274 V=800.0 PL=0
MOVL C01275 V=800.0 PL=0
MOVL C01276 V=800.0 PL=0
MOVL C01277 V=800.0 PL=0
MOVL C01278 V=800.0 PL=0
MOVL C01279 V=800.0 PL=0
MOVL C01280 V=800.0 PL=0
MOVL C01281 V=800.0 PL=0
MOVL C01282 V=800.0 PL=0
MOVL C01283 V=800.0 PL=0
MOVL C01284 V=800.0 PL=0
MOVL C01285 V=800.0 PL=0
MOVL C01286 V=800.0 PL=0
MOVL C01287 V=800.0 PL=0
MOVL C01288 V=800.0 PL=0
MOVL C01289 V=800.0 PL=0
MOVL C01290 V=800.0 PL=0
MOVL C01291 V=800.0 PL=0
MOVL C01292 V=800.0 PL=0
MOVL C01293 V=800.0 PL=0
MOVL C01294 V=800.0 PL=0
MOVL C01295 V=800.0 PL=0
MOVL C01296 V=800.0 PL=0
MOVL C01297 V=800.0 PL=0
MOVL C01298 V=800.0 PL=0
MOVL C01299 V=800.0 PL=0
MOVL C01300 V=800.0 PL=0
MOVL C01301 V=800.0 PL=0
MOVL C01302 V=800.0 PL=0
MOVL C01303 V=800.0 PL=0
MOVL C01304 V=800.0 PL=0
MOVL C01305 V=800.0 PL=0
MOVL C01306 V=800.0 PL=0
MOVL C01307 V=800.0 PL=0
MOVL C01308 V=800.0 PL=0
MOVL C01309 V=800.0 PL=0
MOVL C01310 V=800.0 PL=0
MOVL C01311 V=800.0 PL=0
MOVL C01312 V=800.0 PL=0
MOVL C01313 V=800.0 PL=0
MOVL C01314 V=800.0 PL=0
MOVL C01315 V=800.0 PL=0
MOVL C01316 V=800.0 PL=0
MOVL C01317 V=800.0 PL=0
MOVL C01318 V=800.0 PL=0
MOVL C01319 V=800.0 PL=0
MOVL C01320 V=800.0 PL=0
MOVL C01321 V=800.0 PL=0
MOVL C01322 V=800.0 PL=0
MOVL C01323 V=800.0 PL=0
MOVL C01324 V=800.0 PL=0
MOVL C01325 V=800.0 PL=0
MOVL C01326 V=800.0 PL=0
MOVL C01327 V=800.0 PL=0
MOVL C01328 V=800.0 PL=0
MOVL C01329 V=800.0 PL=0
MOVL C01330 V=800.0 PL=0
MOVL C01331 V=800.0 PL=0
MOVL C01332 V=800.0 PL=0
MOVL C01333 V=800.0 PL=0
MOVL C01334 V=800.0 PL=0
MOVL C01335 V=800.0 PL=0
MOVL C01336 V=800.0 PL=0
MOVL C01337 V=800.0 PL=0
MOVL C01338 V=800.0 PL=0
MOVL C01339 V=800.0 PL=0
MOVL C01340 V=800.0 PL=0
MOVL C01341 V=800.0 PL=0
MOVL C01342 V=800.0 PL=0
MOVL C01343 V=800.0 PL=0
MOVL C01344 V=800.0 PL=0
MOVL C01345 V=800.0 PL=0
MOVL C01346 V=800.0 PL=0
MOVL C01347 V=800.0 PL=0
MOVL C01348 V=800.0 PL=0
MOVL C01349 V=800.0 PL=0
MOVL C01350 V=800.0 PL=0
MOVL C01351 V=800.0 PL=0
MOVL C01352 V=800.0 PL=0
MOVL C01353 V=800.0 PL=0
MOVL C01354 V=800.0 PL=0
MOVL C01355 V=800.0 PL=0
MOVL C01356 V=800.0 PL=0
MOVL C01357 V=800.0 PL=0
MOVL C01358 V=800.0 PL=0
MOVL C01359 V=800.0 PL=0
MOVL C01360 V=800.0 PL=0
MOVL C01361 V=800.0 PL=0
MOVL C01362 V=800.0 PL=0
MOVL C01363 V=800.0 PL=0
MOVL C01364 V=800.0 PL=0
MOVL C01365 V=800.0 PL=0
MOVL C01366 V=800.0 PL=0
MOVL C01367 V=800.0 PL=0
MOVL C01368 V=800.0 PL=0
MOVL C01369 V=800.0 PL=0
MOVL C01370 V=800.0 PL=0
MOVL C01371 V=800.0 PL=0
MOVL C01372 V=800.0 PL=0
MOVL C01373 V=800.0 PL=0
MOVL C01374 V=800.0 PL=0
MOVL C01375 V=800.0 PL=0
MOVL C01376 V=800.0 PL=0
MOVL C01377 V=800.0 PL=0
MOVL C01378 V=800.0 PL=0
MOVL C01379 V=800.0 PL=0
MOVL C01380 V=800.0 PL=0
MOVL C01381 V=800.0 PL=0
MOVL C01382 V=800.0 PL=0
MOVL C01383 V=800.0 PL=0
MOVL C01384 V=800.0 PL=0
MOVL C01385 V=800.0 PL=0
MOVL C01386 V=800.0 PL=0
MOVL C01387 V=800.0 PL=0
MOVL C01388 V=800.0 PL=0
MOVL C01389 V=800.0 PL=0
MOVL C01390 V=800.0 PL=0
MOVL C01391 V=800.0 PL=0
MOVL C01392 V=800.0 PL=0
MOVL C01393 V=800.0 PL=0
MOVL C01394 V=800.0 PL=0
MOVL C01395 V=800.0 PL=0
MOVL C01396 V=800.0 PL=0
MOVL C01397 V=800.0 PL=0
MOVL C01398 V=800.0 PL=0
MOVL C01399 V=800.0 PL=0
MOVL C01400 V=800.0 PL=0
MOVL C01401 V=800.0 PL=0
MOVL C01402 V=800.0 PL=0
MOVL C01403 V=800.0 PL=0
MOVL C01404 V=800.0 PL=0
MOVL C01405 V=800.0 PL=0
MOVL C01406 V=800.0 PL=0
MOVL C01407 V=800.0 PL=0
MOVL C01408 V=800.0 PL=0
MOVL C01409 V=800.0 PL=0
MOVL C01410 V=800.0 PL=0
MOVL C01411 V=800.0 PL=0
MOVL C01412 V=800.0 PL=0
MOVL C01413 V=800.0 PL=0
MOVL C01414 V=800.0 PL=0
MOVL C01415 V=800.0 PL=0
MOVL C01416 V=800.0 PL=0
MOVL C01417 V=800.0 PL=0
MOVL C01418 V=800.0 PL=0
MOVL C01419 V=800.0 PL=0
MOVL C01420 V=800.0 PL=0
MOVL C01421 V=800.0 PL=0
MOVL C01422 V=800.0 PL=0
MOVL C01423 V=800.0 PL=0
MOVL C01424 V=800.0 PL=0
MOVL C01425 V=800.0 PL=0
MOVL C01426 V=800.0 PL=0
MOVL C01427 V=800.0 PL=0
MOVL C01428 V=800.0 PL=0
MOVL C01429 V=800.0 PL=0
MOVL C01430 V=800.0 PL=0
MOVL C01431 V=800.0 PL=0
MOVL C01432 V=800.0 PL=0
MOVL C01433 V=800.0 PL=0
MOVL C01434 V=800.0 PL=0
MOVL C01435 V=800.0 PL=0
MOVL C01436 V=800.0 PL=0
MOVL C01437 V=800.0 PL=0
MOVL C01438 V=800.0 PL=0
MOVL C01439 V=800.0 PL=0
MOVL C01440 V=800.0 PL=0
MOVL C01441 V=800.0 PL=0
MOVL C01442 V=800.0 PL=0
MOVL C01443 V=800.0 PL=0
MOVL C01444 V=800.0 PL=0
MOVL C01445 V=800.0 PL=0
MOVL C01446 V=800.0 PL=0
MOVL C01447 V=800.0 PL=0
MOVL C01448 V=800.0 PL=0
MOVL C01449 V=800.0 PL=0
MOVL C01450 V=800.0 PL=0
MOVL C01451 V=800.0 PL=0
MOVL C01452 V=800.0 PL=0
MOVL C01453 V=800.0 PL=0
MOVL C01454 V=800.0 PL=0
MOVL C01455 V=800.0 PL=0
MOVL C01456 V=800.0 PL=0
MOVL C01457 V=800.0 PL=0
MOVL C01458 V=800.0 PL=0
MOVL C01459 V=800.0 PL=0
MOVL C01460 V=800.0 PL=0
MOVL C01461 V=800.0 PL=0
MOVL C01462 V=800.0 PL=0
MOVL C01463 V=800.0 PL=0
MOVL C01464 V=800.0 PL=0
MOVL C01465 V=800.0 PL=0
MOVL C01466 V=800.0 PL=0
MOVL C01467 V=800.0 PL=0
MOVL C01468 V=800.0 PL=0
MOVL C01469 V=800.0 PL=0
MOVL C01470 V=800.0 PL=0
MOVL C01471 V=800.0 PL=0
MOVL C01472 V=800.0 PL=0
MOVL C01473 V=800.0 PL=0
MOVL C01474 V=800.0 PL=0
MOVL C01475 V=800.0 PL=0
MOVL C01476 V=800.0 PL=0
MOVL C01477 V=800.0 PL=0
MOVL C01478 V=800.0 PL=0
MOVL C01479 V=800.0 PL=0
MOVL C01480 V=800.0 PL=0
MOVL C01481 V=800.0 PL=0
MOVL C01482 V=800.0 PL=0
MOVL C01483 V=800.0 PL=0
MOVL C01484 V=800.0 PL=0
MOVL C01485 V=800.0 PL=0
MOVL C01486 V=800.0 PL=0
MOVL C01487 V=800.0 PL=0
MOVL C01488 V=800.0 PL=0
MOVL C01489 V=800.0 PL=0
MOVL C01490 V=800.0 PL=0
MOVL C01491 V=800.0 PL=0
MOVL C01492 V=800.0 PL=0
MOVL C01493 V=800.0 PL=0
MOVL C01494 V=800.0 PL=0
MOVL C01495 V=800.0 PL=0
MOVL C01496 V=800.0 PL=0
MOVL C01497 V=800.0 PL=0
MOVL C01498 V=800.0 PL=0
MOVL C01499 V=800.0 PL=0
MOVL C01500 V=800.0 PL=0
MOVL C01501 V=800.0 PL=0
MOVL C01502 V=800.0 PL=0
MOVL C01503 V=800.0 PL=0
MOVL C01504 V=800.0 PL=0
MOVL C01505 V=800.0 PL=0
MOVL C01506 V=800.0 PL=0
MOVL C01507 V=800.0 PL=0
MOVL C01508 V=800.0 PL=0
MOVL C01509 V=800.0 PL=0
MOVL C01510 V=800.0 PL=0
MOVL C01511 V=800.0 PL=0
MOVL C01512 V=800.0 PL=0
MOVL C01513 V=800.0 PL=0
MOVL C01514 V=800.0 PL=0
MOVL C01515 V=800.0 PL=0
MOVL C01516 V=800.0 PL=0
MOVL C01517 V=800.0 PL=0
MOVL C01518 V=800.0 PL=0
MOVL C01519 V=800.0 PL=0
MOVL C01520 V=800.0 PL=0
MOVL C01521 V=800.0 PL=0
MOVL C01522 V=800.0 PL=0
MOVL C01523 V=800.0 PL=0
MOVL C01524 V=800.0 PL=0
MOVL C01525 V=800.0 PL=0
MOVL C01526 V=800.0 PL=0
MOVL C01527 V=800.0 PL=0
MOVL C01528 V=800.0 PL=0
MOVL C01529 V=800.0 PL=0
MOVL C01530 V=800.0 PL=0
MOVL C01531 V=800.0 PL=0
MOVL C01532 V=800.0 PL=0
MOVL C01533 V=800.0 PL=0
MOVL C01534 V=800.0 PL=0
MOVL C01535 V=800.0 PL=0
MOVL C01536 V=800.0 PL=0
MOVL C01537 V=800.0 PL=0
MOVL C01538 V=800.0 PL=0
MOVL C01539 V=800.0 PL=0
MOVL C01540 V=800.0 PL=0
MOVL C01541 V=800.0 PL=0
MOVL C01542 V=800.0 PL=0
MOVL C01543 V=800.0 PL=0
MOVL C01544 V=800.0 PL=0
MOVL C01545 V=800.0 PL=0
MOVL C01546 V=800.0 PL=0
MOVL C01547 V=800.0 PL=0
MOVL C01548 V=800.0 PL=0
MOVL C01549 V=800.0 PL=0
MOVL C01550 V=800.0 PL=0
MOVL C01551 V=800.0 PL=0
MOVL C01552 V=800.0 PL=0
MOVL C01553 V=800.0 PL=0
MOVL C01554 V=800.0 PL=0
MOVL C01555 V=800.0 PL=0
MOVL C01556 V=800.0 PL=0
MOVL C01557 V=800.0 PL=0
MOVL C01558 V=800.0 PL=0
MOVL C01559 V=800.0 PL=0
MOVL C01560 V=800.0 PL=0
MOVL C01561 V=800.0 PL=0
MOVL C01562 V=800.0 PL=0
MOVL C01563 V=800.0 PL=0
MOVL C01564 V=800.0 PL=0
MOVL C01565 V=800.0 PL=0
MOVL C01566 V=800.0 PL=0
MOVL C01567 V=800.0 PL=0
MOVL C01568 V=800.0 PL=0
MOVL C01569 V=800.0 PL=0
MOVL C01570 V=800.0 PL=0
MOVL C01571 V=800.0 PL=0
MOVL C01572 V=800.0 PL=0
MOVL C01573 V=800.0 PL=0
MOVL C01574 V=800.0 PL=0
MOVL C01575 V=800.0 PL=0
MOVL C01576 V=800.0 PL=0
MOVL C01577 V=800.0 PL=0
MOVL C01578 V=800.0 PL=0
MOVL C01579 V=800.0 PL=0
MOVL C01580 V=800.0 PL=0
MOVL C01581 V=800.0 PL=0
MOVL C01582 V=800.0 PL=0
MOVL C01583 V=800.0 PL=0
MOVL C01584 V=800.0 PL=0
MOVL C01585 V=800.0 PL=0
MOVL C01586 V=800.0 PL=0
MOVL C01587 V=800.0 PL=0
MOVL C01588 V=800.0 PL=0
MOVL C01589 V=800.0 PL=0
MOVL C01590 V=800.0 PL=0
MOVL C01591 V=800.0 PL=0
MOVL C01592 V=800.0 PL=0
MOVL C01593 V=800.0 PL=0
MOVL C01594 V=800.0 PL=0
MOVL C01595 V=800.0 PL=0
MOVL C01596 V=800.0 PL=0
MOVL C01597 V=800.0 PL=0
MOVL C01598 V=800.0 PL=0
MOVL C01599 V=800.0 PL=0
MOVL C01600 V=800.0 PL=0
MOVL C01601 V=800.0 PL=0
MOVL C01602 V=800.0 PL=0
MOVL C01603 V=800.0 PL=0
MOVL C01604 V=800.0 PL=0
MOVL C01605 V=800.0 PL=0
MOVL C01606 V=800.0 PL=0
MOVL C01607 V=800.0 PL=0
MOVL C01608 V=800.0 PL=0
MOVL C01609 V=800.0 PL=0
MOVL C01610 V=800.0 PL=0
MOVL C01611 V=800.0 PL=0
MOVL C01612 V=800.0 PL=0
MOVL C01613 V=800.0 PL=0
MOVL C01614 V=800.0 PL=0
MOVL C01615 V=800.0 PL=0
MOVL C01616 V=800.0 PL=0
MOVL C01617 V=800.0 PL=0
MOVL C01618 V=800.0 PL=0
MOVL C01619 V=800.0 PL=0
MOVL C01620 V=800.0 PL=0
MOVL C01621 V=800.0 PL=0
MOVL C01622 V=800.0 PL=0
MOVL C01623 V=800.0 PL=0
MOVL C01624 V=800.0 PL=0
MOVL C01625 V=800.0 PL=0
MOVL C01626 V=800.0 PL=0
MOVL C01627 V=800.0 PL=0
MOVL C01628 V=800.0 PL=0
MOVL C01629 V=800.0 PL=0
MOVL C01630 V=800.0 PL=0
MOVL C01631 V=800.0 PL=0
MOVL C01632 V=800.0 PL=0
MOVL C01633 V=800.0 PL=0
MOVL C01634 V=800.0 PL=0
MOVL C01635 V=800.0 PL=0
MOVL C01636 V=800.0 PL=0
MOVL C01637 V=800.0 PL=0
MOVL C01638 V=800.0 PL=0
MOVL C01639 V=800.0 PL=0
MOVL C01640 V=800.0 PL=0
MOVL C01641 V=800.0 PL=0
MOVL C01642 V=800.0 PL=0
MOVL C01643 V=800.0 PL=0
MOVL C01644 V=800.0 PL=0
MOVL C01645 V=800.0 PL=0
MOVL C01646 V=800.0 PL=0
MOVL C01647 V=800.0 PL=0
MOVL C01648 V=800.0 PL=0
MOVL C01649 V=800.0 PL=0
MOVL C01650 V=800.0 PL=0
MOVL C01651 V=800.0 PL=0
MOVL C01652 V=800.0 PL=0
MOVL C01653 V=800.0 PL=0
MOVL C01654 V=800.0 PL=0
MOVL C01655 V=800.0 PL=0
MOVL C01656 V=800.0 PL=0
MOVL C01657 V=800.0 PL=0
MOVL C01658 V=800.0 PL=0
MOVL C01659 V=800.0 PL=0
MOVL C01660 V=800.0 PL=0
MOVL C01661 V=800.0 PL=0
MOVL C01662 V=800.0 PL=0
MOVL C01663 V=800.0 PL=0
MOVL C01664 V=800.0 PL=0
MOVL C01665 V=800.0 PL=0
MOVL C01666 V=800.0 PL=0
MOVL C01667 V=800.0 PL=0
MOVL C01668 V=800.0 PL=0
MOVL C01669 V=800.0 PL=0
MOVL C01670 V=800.0 PL=0
MOVL C01671 V=800.0 PL=0
MOVL C01672 V=800.0 PL=0
MOVL C01673 V=800.0 PL=0
MOVL C01674 V=800.0 PL=0
MOVL C01675 V=800.0 PL=0
MOVL C01676 V=800.0 PL=0
MOVL C01677 V=800.0 PL=0
MOVL C01678 V=800.0 PL=0
MOVL C01679 V=800.0 PL=0
MOVL C01680 V=800.0 PL=0
MOVL C01681 V=800.0 PL=0
MOVL C01682 V=800.0 PL=0
MOVL C01683 V=800.0 PL=0
MOVL C01684 V=800.0 PL=0
MOVL C01685 V=800.0 PL=0
MOVL C01686 V=800.0 PL=0
MOVL C01687 V=800.0 PL=0
MOVL C01688 V=800.0 PL=0
MOVL C01689 V=800.0 PL=0
MOVL C01690 V=800.0 PL=0
MOVL C01691 V=800.0 PL=0
MOVL C01692 V=800.0 PL=0
MOVL C01693 V=800.0 PL=0
MOVL C01694 V=800.0 PL=0
MOVL C01695 V=800.0 PL=0
MOVL C01696 V=800.0 PL=0
MOVL C01697 V=800.0 PL=0
MOVL C01698 V=800.0 PL=0
MOVL C01699 V=800.0 PL=0
MOVL C01700 V=800.0 PL=0
MOVL C01701 V=800.0 PL=0
MOVL C01702 V=800.0 PL=0
MOVL C01703 V=800.0 PL=0
MOVL C01704 V=800.0 PL=0
MOVL C01705 V=800.0 PL=0
MOVL C01706 V=800.0 PL=0
MOVL C01707 V=800.0 PL=0
MOVL C01708 V=800.0 PL=0
MOVL C01709 V=800.0 PL=0
MOVL C01710 V=800.0 PL=0
MOVL C01711 V=800.0 PL=0
MOVL C01712 V=800.0 PL=0
MOVL C01713 V=800.0 PL=0
MOVL C01714 V=800.0 PL=0
MOVL C01715 V=800.0 PL=0
MOVL C01716 V=800.0 PL=0
MOVL C01717 V=800.0 PL=0
MOVL C01718 V=800.0 PL=0
MOVL C01719 V=800.0 PL=0
MOVL C01720 V=800.0 PL=0
MOVL C01721 V=800.0 PL=0
MOVL C01722 V=800.0 PL=0
MOVL C01723 V=800.0 PL=0
MOVL C01724 V=800.0 PL=0
MOVL C01725 V=800.0 PL=0
MOVL C01726 V=800.0 PL=0
MOVL C01727 V=800.0 PL=0
MOVL C01728 V=800.0 PL=0
MOVL C01729 V=800.0 PL=0
MOVL C01730 V=800.0 PL=0
MOVL C01731 V=800.0 PL=0
MOVL C01732 V=800.0 PL=0
MOVL C01733 V=800.0 PL=0
MOVL C01734 V=800.0 PL=0
MOVL C01735 V=800.0 PL=0
MOVL C01736 V=800.0 PL=0
MOVL C01737 V=800.0 PL=0
MOVL C01738 V=800.0 PL=0
MOVL C01739 V=800.0 PL=0
MOVL C01740 V=800.0 PL=0
MOVL C01741 V=800.0 PL=0
MOVL C01742 V=800.0 PL=0
MOVL C01743 V=800.0 PL=0
MOVL C01744 V=800.0 PL=0
MOVL C01745 V=800.0 PL=0
MOVL C01746 V=800.0 PL=0
MOVL C01747 V=800.0 PL=0
MOVL C01748 V=800.0 PL=0
MOVL C01749 V=800.0 PL=0
MOVL C01750 V=800.0 PL=0
MOVL C01751 V=800.0 PL=0
MOVL C01752 V=800.0 PL=0
MOVL C01753 V=800.0 PL=0
MOVL C01754 V=800.0 PL=0
MOVL C01755 V=800.0 PL=0
MOVL C01756 V=800.0 PL=0
MOVL C01757 V=800.0 PL=0
MOVL C01758 V=800.0 PL=0
MOVL C01759 V=800.0 PL=0
MOVL C01760 V=800.0 PL=0
MOVL C01761 V=800.0 PL=0
MOVL C01762 V=800.0 PL=0
MOVL C01763 V=800.0 PL=0
MOVL C01764 V=800.0 PL=0
MOVL C01765 V=800.0 PL=0
MOVL C01766 V=800.0 PL=0
MOVL C01767 V=800.0 PL=0
MOVL C01768 V=800.0 PL=0
MOVL C01769 V=800.0 PL=0
MOVL C01770 V=800.0 PL=0
MOVL C01771 V=800.0 PL=0
MOVL C01772 V=800.0 PL=0
MOVL C01773 V=800.0 PL=0
MOVL C01774 V=800.0 PL=0
MOVL C01775 V=800.0 PL=0
MOVL C01776 V=800.0 PL=0
MOVL C01777 V=800.0 PL=0
MOVL C01778 V=800.0 PL=0
MOVL C01779 V=800.0 PL=0
MOVL C01780 V=800.0 PL=0
MOVL C01781 V=800.0 PL=0
MOVL C01782 V=800.0 PL=0
MOVL C01783 V=800.0 PL=0
MOVL C01784 V=800.0 PL=0
MOVL C01785 V=800.0 PL=0
MOVL C01786 V=800.0 PL=0
MOVL C01787 V=800.0 PL=0
MOVL C01788 V=800.0 PL=0
MOVL C01789 V=800.0 PL=0
MOVL C01790 V=800.0 PL=0
MOVL C01791 V=800.0 PL=0
MOVL C01792 V=800.0 PL=0
MOVL C01793 V=800.0 PL=0
MOVL C01794 V=800.0 PL=0
MOVL C01795 V=800.0 PL=0
MOVL C01796 V=800.0 PL=0
MOVL C01797 V=800.0 PL=0
MOVL C01798 V=800.0 PL=0
MOVL C01799 V=800.0 PL=0
MOVL C01800 V=800.0 PL=0
MOVL C01801 V=800.0 PL=0
MOVL C01802 V=800.0 PL=0
MOVL C01803 V=800.0 PL=0
MOVL C01804 V=800.0 PL=0
MOVL C01805 V=800.0 PL=0
MOVL C01806 V=800.0 PL=0
MOVL C01807 V=800.0 PL=0
MOVL C01808 V=800.0 PL=0
MOVL C01809 V=800.0 PL=0
MOVL C01810 V=800.0 PL=0
MOVL C01811 V=800.0 PL=0
MOVL C01812 V=800.0 PL=0
MOVL C01813 V=800.0 PL=0
MOVL C01814 V=800.0 PL=0
MOVL C01815 V=800.0 PL=0
MOVL C01816 V=800.0 PL=0
MOVL C01817 V=800.0 PL=0
MOVL C01818 V=800.0 PL=0
MOVL C01819 V=800.0 PL=0
MOVL C01820 V=800.0 PL=0
MOVL C01821 V=800.0 PL=0
MOVL C01822 V=800.0 PL=0
MOVL C01823 V=800.0 PL=0
MOVL C01824 V=800.0 PL=0
MOVL C01825 V=800.0 PL=0
MOVL C01826 V=800.0 PL=0
MOVL C01827 V=800.0 PL=0
MOVL C01828 V=800.0 PL=0
MOVL C01829 V=800.0 PL=0
MOVL C01830 V=800.0 PL=0
MOVL C01831 V=800.0 PL=0
MOVL C01832 V=800.0 PL=0
MOVL C01833 V=800.0 PL=0
MOVL C01834 V=800.0 PL=0
MOVL C01835 V=800.0 PL=0
MOVL C01836 V=800.0 PL=0
MOVL C01837 V=800.0 PL=0
MOVL C01838 V=800.0 PL=0
MOVL C01839 V=800.0 PL=0
MOVL C01840 V=800.0 PL=0
MOVL C01841 V=800.0 PL=0
MOVL C01842 V=800.0 PL=0
MOVL C01843 V=800.0 PL=0
MOVL C01844 V=800.0 PL=0
MOVL C01845 V=800.0 PL=0
MOVL C01846 V=800.0 PL=0
MOVL C01847 V=800.0 PL=0
MOVL C01848 V=800.0 PL=0
MOVL C01849 V=800.0 PL=0
MOVL C01850 V=800.0 PL=0
MOVL C01851 V=800.0 PL=0
MOVL C01852 V=800.0 PL=0
MOVL C01853 V=800.0 PL=0
MOVL C01854 V=800.0 PL=0
MOVL C01855 V=800.0 PL=0
MOVL C01856 V=800.0 PL=0
MOVL C01857 V=800.0 PL=0
MOVL C01858 V=800.0 PL=0
MOVL C01859 V=800.0 PL=0
MOVL C01860 V=800.0 PL=0
MOVL C01861 V=800.0 PL=0
MOVL C01862 V=800.0 PL=0
MOVL C01863 V=800.0 PL=0
MOVL C01864 V=800.0 PL=0
MOVL C01865 V=800.0 PL=0
MOVL C01866 V=800.0 PL=0
MOVL C01867 V=800.0 PL=0
MOVL C01868 V=800.0 PL=0
MOVL C01869 V=800.0 PL=0
MOVL C01870 V=800.0 PL=0
MOVL C01871 V=800.0 PL=0
MOVL C01872 V=800.0 PL=0
MOVL C01873 V=800.0 PL=0
MOVL C01874 V=800.0 PL=0
MOVL C01875 V=800.0 PL=0
MOVL C01876 V=800.0 PL=0
MOVL C01877 V=800.0 PL=0
MOVL C01878 V=800.0 PL=0
MOVL C01879 V=800.0 PL=0
MOVL C01880 V=800.0 PL=0
MOVL C01881 V=800.0 PL=0
MOVL C01882 V=800.0 PL=0
MOVL C01883 V=800.0 PL=0
MOVL C01884 V=800.0 PL=0
MOVL C01885 V=800.0 PL=0
MOVL C01886 V=800.0 PL=0
MOVL C01887 V=800.0 PL=0
MOVL C01888 V=800.0 PL=0
MOVL C01889 V=800.0 PL=0
MOVL C01890 V=800.0 PL=0
MOVL C01891 V=800.0 PL=0
MOVL C01892 V=800.0 PL=0
MOVL C01893 V=800.0 PL=0
MOVL C01894 V=800.0 PL=0
MOVL C01895 V=800.0 PL=0
MOVL C01896 V=800.0 PL=0
MOVL C01897 V=800.0 PL=0
MOVL C01898 V=800.0 PL=0
MOVL C01899 V=800.0 PL=0
MOVL C01900 V=800.0 PL=0
MOVL C01901 V=800.0 PL=0
MOVL C01902 V=800.0 PL=0
MOVL C01903 V=800.0 PL=0
MOVL C01904 V=800.0 PL=0
MOVL C01905 V=800.0 PL=0
MOVL C01906 V=800.0 PL=0
MOVL C01907 V=800.0 PL=0
MOVL C01908 V=800.0 PL=0
MOVL C01909 V=800.0 PL=0
MOVL C01910 V=800.0 PL=0
MOVL C01911 V=800.0 PL=0
MOVL C01912 V=800.0 PL=0
MOVL C01913 V=800.0 PL=0
MOVL C01914 V=800.0 PL=0
MOVL C01915 V=800.0 PL=0
MOVL C01916 V=800.0 PL=0
MOVL C01917 V=800.0 PL=0
MOVL C01918 V=800.0 PL=0
MOVL C01919 V=800.0 PL=0
MOVL C01920 V=800.0 PL=0
MOVL C01921 V=800.0 PL=0
MOVL C01922 V=800.0 PL=0
MOVL C01923 V=800.0 PL=0
MOVL C01924 V=800.0 PL=0
MOVL C01925 V=800.0 PL=0
MOVL C01926 V=800.0 PL=0
MOVL C01927 V=800.0 PL=0
MOVL C01928 V=800.0 PL=0
MOVL C01929 V=800.0 PL=0
MOVL C01930 V=800.0 PL=0
MOVL C01931 V=800.0 PL=0
MOVL C01932 V=800.0 PL=0
MOVL C01933 V=800.0 PL=0
MOVL C01934 V=800.0 PL=0
MOVL C01935 V=800.0 PL=0
MOVL C01936 V=800.0 PL=0
MOVL C01937 V=800.0 PL=0
MOVL C01938 V=800.0 PL=0
MOVL C01939 V=800.0 PL=0
MOVL C01940 V=800.0 PL=0
MOVL C01941 V=800.0 PL=0
MOVL C01942 V=800.0 PL=0
MOVL C01943 V=800.0 PL=0
MOVL C01944 V=800.0 PL=0
MOVL C01945 V=800.0 PL=0
MOVL C01946 V=800.0 PL=0
MOVL C01947 V=800.0 PL=0
MOVL C01948 V=800.0 PL=0
MOVL C01949 V=800.0 PL=0
MOVL C01950 V=800.0 PL=0
MOVL C01951 V=800.0 PL=0
MOVL C01952 V=800.0 PL=0
MOVL C01953 V=800.0 PL=0
MOVL C01954 V=800.0 PL=0
MOVL C01955 V=800.0 PL=0
MOVL C01956 V=800.0 PL=0
MOVL C01957 V=800.0 PL=0
MOVL C01958 V=800.0 PL=0
MOVL C01959 V=800.0 PL=0
MOVL C01960 V=800.0 PL=0
MOVL C01961 V=800.0 PL=0
MOVL C01962 V=800.0 PL=0
MOVL C01963 V=800.0 PL=0
MOVL C01964 V=800.0 PL=0
MOVL C01965 V=800.0 PL=0
MOVL C01966 V=800.0 PL=0
MOVL C01967 V=800.0 PL=0
MOVL C01968 V=800.0 PL=0
MOVL C01969 V=800.0 PL=0
MOVL C01970 V=800.0 PL=0
MOVL C01971 V=800.0 PL=0
MOVL C01972 V=800.0 PL=0
MOVL C01973 V=800.0 PL=0
MOVL C01974 V=800.0 PL=0
MOVL C01975 V=800.0 PL=0
MOVL C01976 V=800.0 PL=0
MOVL C01977 V=800.0 PL=0
MOVL C01978 V=800.0 PL=0
MOVL C01979 V=800.0 PL=0
MOVL C01980 V=800.0 PL=0
MOVL C01981 V=800.0 PL=0
MOVL C01982 V=800.0 PL=0
MOVL C01983 V=800.0 PL=0
MOVL C01984 V=800.0 PL=0
MOVL C01985 V=800.0 PL=0
MOVL C01986 V=800.0 PL=0
MOVL C01987 V=800.0 PL=0
MOVL C01988 V=800.0 PL=0
MOVL C01989 V=800.0 PL=0
MOVL C01990 V=800.0 PL=0
MOVL C01991 V=800.0 PL=0
MOVL C01992 V=800.0 PL=0
MOVL C01993 V=800.0 PL=0
MOVL C01994 V=800.0 PL=0
MOVL C01995 V=800.0 PL=0
MOVL C01996 V=800.0 PL=0
MOVL C01997 V=800.0 PL=0
MOVL C01998 V=800.0 PL=0
MOVL C01999 V=800.0 PL=0
MOVL C02000 V=800.0 PL=0
MOVL C02001 V=800.0 PL=0
MOVL C02002 V=800.0 PL=0
MOVL C02003 V=800.0 PL=0
MOVL C02004 V=800.0 PL=0
MOVL C02005 V=800.0 PL=0
MOVL C02006 V=800.0 PL=0
MOVL C02007 V=800.0 PL=0
MOVL C02008 V=800.0 PL=0
MOVL C02009 V=800.0 PL=0
MOVL C02010 V=800.0 PL=0
MOVL C02011 V=800.0 PL=0
MOVL C02012 V=800.0 PL=0
MOVL C02013 V=800.0 PL=0
MOVL C02014 V=800.0 PL=0
MOVL C02015 V=800.0 PL=0
MOVL C02016 V=800.0 PL=0
MOVL C02017 V=800.0 PL=0
MOVL C02018 V=800.0 PL=0
MOVL C02019 V=800.0 PL=0
MOVL C02020 V=800.0 PL=0
MOVL C02021 V=800.0 PL=0
MOVL C02022 V=800.0 PL=0
MOVL C02023 V=800.0 PL=0
MOVL C02024 V=800.0 PL=0
MOVL C02025 V=800.0 PL=0
MOVL C02026 V=800.0 PL=0
MOVL C02027 V=800.0 PL=0
MOVL C02028 V=800.0 PL=0
MOVL C02029 V=800.0 PL=0
MOVL C02030 V=800.0 PL=0
MOVL C02031 V=800.0 PL=0
MOVL C02032 V=800.0 PL=0
MOVL C02033 V=800.0 PL=0
MOVL C02034 V=800.0 PL=0
MOVL C02035 V=800.0 PL=0
MOVL C02036 V=800.0 PL=0
MOVL C02037 V=800.0 PL=0
MOVL C02038 V=800.0 PL=0
MOVL C02039 V=800.0 PL=0
MOVL C02040 V=800.0 PL=0
MOVL C02041 V=800.0 PL=0
MOVL C02042 V=800.0 PL=0
MOVL C02043 V=800.0 PL=0
MOVL C02044 V=800.0 PL=0
MOVL C02045 V=800.0 PL=0
MOVL C02046 V=800.0 PL=0
MOVL C02047 V=800.0 PL=0
MOVL C02048 V=800.0 PL=0
MOVL C02049 V=800.0 PL=0
MOVL C02050 V=800.0 PL=0
MOVL C02051 V=800.0 PL=0
MOVL C02052 V=800.0 PL=0
MOVL C02053 V=800.0 PL=0
MOVL C02054 V=800.0 PL=0
MOVL C02055 V=800.0 PL=0
MOVL C02056 V=800.0 PL=0
MOVL C02057 V=800.0 PL=0
MOVL C02058 V=800.0 PL=0
MOVL C02059 V=800.0 PL=0
MOVL C02060 V=800.0 PL=0
MOVL C02061 V=800.0 PL=0
MOVL C02062 V=800.0 PL=0
MOVL C02063 V=800.0 PL=0
MOVL C02064 V=800.0 PL=0
MOVL C02065 V=800.0 PL=0
MOVL C02066 V=800.0 PL=0
MOVL C02067 V=800.0 PL=0
MOVL C02068 V=800.0 PL=0
MOVL C02069 V=800.0 PL=0
MOVL C02070 V=800.0 PL=0
MOVL C02071 V=800.0 PL=0
MOVL C02072 V=800.0 PL=0
MOVL C02073 V=800.0 PL=0
MOVL C02074 V=800.0 PL=0
MOVL C02075 V=800.0 PL=0
MOVL C02076 V=800.0 PL=0
MOVL C02077 V=800.0 PL=0
MOVL C02078 V=800.0 PL=0
MOVL C02079 V=800.0 PL=0
MOVL C02080 V=800.0 PL=0
MOVL C02081 V=800.0 PL=0
MOVL C02082 V=800.0 PL=0
MOVL C02083 V=800.0 PL=0
MOVL C02084 V=800.0 PL=0
MOVL C02085 V=800.0 PL=0
MOVL C02086 V=800.0 PL=0
MOVL C02087 V=800.0 PL=0
MOVL C02088 V=800.0 PL=0
MOVL C02089 V=800.0 PL=0
MOVL C02090 V=800.0 PL=0
MOVL C02091 V=800.0 PL=0
MOVL C02092 V=800.0 PL=0
MOVL C02093 V=800.0 PL=0
MOVL C02094 V=800.0 PL=0
MOVL C02095 V=800.0 PL=0
MOVL C02096 V=800.0 PL=0
MOVL C02097 V=800.0 PL=0
MOVL C02098 V=800.0 PL=0
MOVL C02099 V=800.0 PL=0
MOVL C02100 V=800.0 PL=0
MOVL C02101 V=800.0 PL=0
MOVL C02102 V=800.0 PL=0
MOVL C02103 V=800.0 PL=0
MOVL C02104 V=800.0 PL=0
MOVL C02105 V=800.0 PL=0
MOVL C02106 V=800.0 PL=0
MOVL C02107 V=800.0 PL=0
MOVL C02108 V=800.0 PL=0
MOVL C02109 V=800.0 PL=0
